  MoveL 2858 to (545.28, 463.11, 48) mm, rotated rx -180 ry 0 rz 160 deg; joints [1.397, 78.332, -23.257, -154.456, 57.789, 165.708]
  Call Extruder(423.12650)
  MoveL 2859 to (546.03, 464.05, 48) mm, rotated rx 180 ry 0 rz 160 deg; joints [1.504, 78.485, -23.584, -154.287, 57.658, 165.554]
  Set speed (17.6 mm/s)
  Call Extruder(426.93166)
  MoveL 2860 to (546.75, 464.99, 48) mm, rotated rx -180 ry 0 rz 160 deg; joints [1.61, 78.632, -23.9, -154.118, 57.533, 165.401]
  Set speed (17.6 mm/s)
  Call Extruder(430.87800)
  MoveL 2861 to (547.48, 465.98, 48) mm, rotated rx 180 ry 0 rz 160 deg; joints [1.722, 78.782, -24.221, -153.941, 57.407, 165.243]
  Set speed (17.6 mm/s)
  Call Extruder(434.56337)
  MoveL 2862 to (548.14, 466.92, 48) mm, rotated rx 180 ry 0 rz 160 deg; joints [1.828, 78.92, -24.516, -153.776, 57.293, 165.095]
  Set speed (17.6 mm/s)
  Call Extruder(438.45260)
  MoveL 2863 to (548.81, 467.93, 48) mm, rotated rx -180 ry 0 rz 160 deg; joints [1.941, 79.062, -24.821, -153.599, 57.177, 164.94]
  Set speed (17.6 mm/s)
  Call Extruder(442.25039)
  MoveL 2864 to (549.45, 468.92, 48) mm, rotated rx -180 ry 0 rz 160 deg; joints [2.053, 79.2, -25.114, -153.426, 57.067, 164.787]
  Set speed (17.6 mm/s)
  Call Extruder(446.16761)
  MoveL 2865 to (550.09, 469.96, 48) mm, rotated rx 180 ry 0 rz 160 deg; joints [2.17, 79.337, -25.408, -153.247, 56.958, 164.631]
  Set speed (17.6 mm/s)
  Call Extruder(449.89930)
  MoveL 2866 to (550.68, 470.96, 48) mm, rotated rx 180 ry 0 rz 160 deg; joints [2.282, 79.467, -25.683, -153.075, 56.857, 164.481]
  Set speed (17.6 mm/s)
  Call Extruder(454.87335)
  MoveL 2867 to (551.43, 472.32, 48) mm, rotated rx -180 ry 0 rz 160 deg; joints [2.433, 79.634, -26.039, -152.844, 56.73, 164.284]
  Call Extruder(457.60694)
  MoveL 2868 to (551.83, 473.07, 48) mm, rotated rx -180 ry 0 rz 160 deg; joints [2.517, 79.723, -26.229, -152.717, 56.664, 164.175]
  Set speed (17.6 mm/s)
  Call Extruder(461.47028)
  MoveL 2869 to (552.38, 474.15, 48) mm, rotated rx -180 ry 0 rz 160 deg; joints [2.637, 79.847, -26.493, -152.537, 56.572, 164.023]
  Call Extruder(465.26660)
  MoveL 2870 to (552.89, 475.21, 48) mm, rotated rx -180 ry 0 rz 160 deg; joints [2.756, 79.966, -26.744, -152.36, 56.487, 163.873]
  Call Extruder(469.15969)
  MoveL 2871 to (553.39, 476.32, 48) mm, rotated rx 180 ry 0 rz 160 deg; joints [2.878, 80.083, -26.994, -152.177, 56.405, 163.721]
  Set speed (17.6 mm/s)
  Call Extruder(473.03101)
  MoveL 2872 to (553.87, 477.43, 48) mm, rotated rx -180 ry 0 rz 160 deg; joints [3.002, 80.196, -27.233, -151.996, 56.328, 163.572]
  Set speed (17.6 mm/s)
  Call Extruder(476.66330)
  MoveL 2873 to (554.3, 478.47, 48) mm, rotated rx -180 ry 0 rz 160 deg; joints [3.118, 80.3, -27.453, -151.826, 56.258, 163.432]
  Set speed (17.6 mm/s)
  Call Extruder(484.36900)
  MoveL 2874 to (555.14, 480.72, 48) mm, rotated rx 180 ry 0 rz 160 deg; joints [3.367, 80.508, -27.894, -151.464, 56.126, 163.139]
  Set speed (17.6 mm/s)
  Call Extruder(488.35091)
  MoveL 2875 to (555.53, 481.9, 48) mm, rotated rx -180 ry 0 rz 160 deg; joints [3.498, 80.609, -28.106, -151.278, 56.066, 162.991]
  Set speed (17.6 mm/s)
  Call Extruder(492.11041)
  MoveL 2876 to (555.88, 483.01, 48) mm, rotated rx -180 ry 0 rz 160 deg; joints [3.621, 80.701, -28.301, -151.102, 56.012, 162.851]
  Call Extruder(496.03639)
  MoveL 2877 to (556.22, 484.19, 48) mm, rotated rx -180 ry 0 rz 160 deg; joints [3.751, 80.792, -28.492, -150.919, 55.962, 162.709]
  Set speed (17.6 mm/s)
  Call Extruder(499.92428)
  MoveL 2878 to (556.54, 485.35, 48) mm, rotated rx -180 ry 0 rz 160 deg; joints [3.881, 80.879, -28.677, -150.738, 55.916, 162.568]
  Set speed (17.6 mm/s)
  Call Extruder(507.43789)
  MoveL 2879 to (557.09, 487.63, 48) mm, rotated rx -180 ry 0 rz 160 deg; joints [4.133, 81.034, -29.003, -150.391, 55.843, 162.303]
  Set speed (17.6 mm/s)
  Call Extruder(515.16993)
  MoveL 2880 to (557.55, 490, 48) mm, rotated rx -180 ry 0 rz 160 deg; joints [4.395, 81.176, -29.302, -150.036, 55.787, 162.039]
  Set speed (17.6 mm/s)
  Call Extruder(522.84550)
  MoveL 2881 to (557.91, 492.36, 48) mm, rotated rx -180 ry 0 rz 160 deg; joints [4.658, 81.298, -29.56, -149.688, 55.751, 161.788]
  Set speed (17.6 mm/s)
  Call Extruder(530.59967)
  MoveL 2882 to (558.17, 494.77, 48) mm, rotated rx -180 ry 0 rz 160 deg; joints [4.924, 81.404, -29.781, -149.341, 55.735, 161.544]
  Set speed (17.6 mm/s)
  Call Extruder(538.17218)
  MoveL 2883 to (558.34, 497.12, 48) mm, rotated rx 180 ry 0 rz 160 deg; joints [5.187, 81.488, -29.957, -149.008, 55.74, 161.317]
  Set speed (17.6 mm/s)
  Call Extruder(545.84219)
  MoveL 2884 to (558.41, 499.51, 48) mm, rotated rx 180 ry 0 rz 160 deg; joints [5.453, 81.553, -30.096, -148.677, 55.764, 161.1]
  Set speed (17.6 mm/s)
  Call Extruder(553.37640)
  MoveL 2885 to (558.38, 501.86, 48) mm, rotated rx -180 ry 0 rz 160 deg; joints [5.716, 81.599, -30.192, -148.359, 55.806, 160.899]
  Set speed (17.6 mm/s)
  Call Extruder(561.15643)
  MoveL 2886 to (558.25, 504.28, 48) mm, rotated rx -180 ry 0 rz 160 deg; joints [5.988, 81.627, -30.25, -148.038, 55.87, 160.705]
  Set speed (17.6 mm/s)
  Call Extruder(568.72691)
  MoveL 2887 to (558.03, 506.63, 48) mm, rotated rx 180 ry 0 rz 160 deg; joints [6.253, 81.634, -30.264, -147.733, 55.951, 160.531]
  Set speed (17.6 mm/s)
  Call Extruder(576.57629)
  MoveL 2888 to (557.7, 509.06, 48) mm, rotated rx -180 ry 0 rz 160 deg; joints [6.528, 81.621, -30.238, -147.426, 56.055, 160.366]
  Set speed (17.6 mm/s)
  Call Extruder(584.14957)
  MoveL 2889 to (557.29, 511.38, 48) mm, rotated rx -180 ry 0 rz 160 deg; joints [6.793, 81.589, -30.17, -147.139, 56.174, 160.221]
  Set speed (17.6 mm/s)
  Call Extruder(591.90187)
  MoveL 2890 to (556.77, 513.74, 48) mm, rotated rx -180 ry 0 rz 160 deg; joints [7.063, 81.537, -30.061, -146.854, 56.314, 160.089]
  Call Extruder(599.47109)
  MoveL 2891 to (556.17, 516.02, 48) mm, rotated rx -180 ry 0 rz 160 deg; joints [7.326, 81.466, -29.912, -146.585, 56.469, 159.976]
  Set speed (17.6 mm/s)
  Call Extruder(602.44592)
  MoveL 2892 to (555.91, 516.91, 48) mm, rotated rx 180 ry 0 rz 160 deg; joints [7.429, 81.432, -29.841, -146.483, 56.535, 159.937]
  Set speed (17.6 mm/s)
  Call Extruder(607.08358)
  MoveL 2893 to (555.47, 518.29, 48) mm, rotated rx 180 ry 0 rz 160 deg; joints [7.588, 81.376, -29.722, -146.326, 56.642, 159.879]
  Set speed (17.6 mm/s)
  Call Extruder(614.72062)
  MoveL 2894 to (554.68, 520.53, 48) mm, rotated rx 180 ry 0 rz 160 deg; joints [7.851, 81.267, -29.494, -146.075, 56.832, 159.797]
  Set speed (17.6 mm/s)
  Call Extruder(618.66676)
  MoveL 2895 to (554.23, 521.68, 48) mm, rotated rx -180 ry 0 rz 160 deg; joints [7.986, 81.203, -29.358, -145.95, 56.937, 159.762]
  Set speed (17.6 mm/s)
  Call Extruder(622.59881)
  MoveL 2896 to (553.77, 522.81, 48) mm, rotated rx -180 ry 0 rz 160 deg; joints [8.12, 81.136, -29.218, -145.827, 57.044, 159.73]
  Set speed (17.6 mm/s)
  Call Extruder(626.34222)
  MoveL 2897 to (553.3, 523.88, 48) mm, rotated rx -180 ry 0 rz 160 deg; joints [8.246, 81.066, -29.07, -145.714, 57.152, 159.705]
  Set speed (17.6 mm/s)
  Call Extruder(630.01061)
  MoveL 2898 to (552.83, 524.92, 48) mm, rotated rx -180 ry 0 rz 160 deg; joints [8.37, 80.995, -28.921, -145.604, 57.26, 159.683]
  Set speed (17.6 mm/s)
  Call Extruder(634.07248)
  MoveL 2899 to (552.27, 526.06, 48) mm, rotated rx -180 ry 0 rz 160 deg; joints [8.506, 80.912, -28.745, -145.486, 57.384, 159.663]
  Set speed (17.6 mm/s)
  Call Extruder(638.12886)
  MoveL 2900 to (551.7, 527.18, 48) mm, rotated rx -180 ry 0 rz 160 deg; joints [8.642, 80.823, -28.559, -145.371, 57.512, 159.648]
  Call Extruder(641.69777)
  MoveL 2901 to (551.17, 528.16, 48) mm, rotated rx 180 ry 0 rz 160 deg; joints [8.76, 80.741, -28.385, -145.272, 57.628, 159.639]
  Set speed (17.6 mm/s)
  Call Extruder(645.41195)
  MoveL 2902 to (550.6, 529.17, 48) mm, rotated rx -180 ry 0 rz 160 deg; joints [8.883, 80.652, -28.198, -145.171, 57.752, 159.633]
  Set speed (17.6 mm/s)
  Call Extruder(649.34423)
  MoveL 2903 to (549.98, 530.23, 48) mm, rotated rx -180 ry 0 rz 160 deg; joints [9.012, 80.554, -27.991, -145.068, 57.886, 159.63]
  Set speed (17.6 mm/s)
  Call Extruder(653.08075)
  MoveL 2904 to (549.37, 531.22, 48) mm, rotated rx 180 ry 0 rz 160 deg; joints [9.134, 80.457, -27.785, -144.972, 58.017, 159.632]
  Set speed (17.6 mm/s)
  Call Extruder(656.63345)
  MoveL 2905 to (548.77, 532.15, 48) mm, rotated rx -180 ry 0 rz 160 deg; joints [9.249, 80.361, -27.582, -144.883, 58.145, 159.637]
  Set speed (17.6 mm/s)
  Call Extruder(660.74663)
  MoveL 2906 to (548.05, 533.21, 48) mm, rotated rx 180 ry 0 rz 160 deg; joints [9.382, 80.245, -27.338, -144.783, 58.297, 159.648]
  Set speed (17.6 mm/s)
  Call Extruder(664.63531)
  MoveL 2907 to (547.35, 534.2, 48) mm, rotated rx -180 ry 0 rz 160 deg; joints [9.506, 80.133, -27.1, -144.691, 58.442, 159.661]
  Set speed (17.6 mm/s)
  Call Extruder(668.54814)
  MoveL 2908 to (546.62, 535.19, 48) mm, rotated rx 180 ry 0 rz 160 deg; joints [9.63, 80.017, -26.853, -144.601, 58.592, 159.678]
  Call Extruder(672.23601)
  MoveL 2909 to (545.92, 536.1, 48) mm, rotated rx -180 ry 0 rz 160 deg; joints [9.746, 79.903, -26.611, -144.519, 58.736, 159.699]
  Set speed (17.6 mm/s)
  Call Extruder(676.15166)
  MoveL 2910 to (545.16, 537.05, 48) mm, rotated rx -180 ry 0 rz 160 deg; joints [9.868, 79.779, -26.348, -144.434, 58.892, 159.724]
  Call Extruder(679.91758)
  MoveL 2911 to (544.4, 537.95, 48) mm, rotated rx -180 ry 0 rz 160 deg; joints [9.984, 79.656, -26.087, -144.355, 59.044, 159.753]
  Set speed (17.6 mm/s)
  Call Extruder(683.75230)
  MoveL 2912 to (543.62, 538.85, 48) mm, rotated rx 180 ry 0 rz 160 deg; joints [10.101, 79.528, -25.815, -144.278, 59.202, 159.785]
  Call Extruder(687.54414)
  MoveL 2913 to (542.82, 539.72, 48) mm, rotated rx 180 ry 0 rz 160 deg; joints [10.216, 79.399, -25.54, -144.203, 59.36, 159.82]
  Set speed (17.6 mm/s)
  Call Extruder(690.70425)
  MoveL 2914 to (542.15, 540.44, 48) mm, rotated rx 180 ry 0 rz 160 deg; joints [10.31, 79.289, -25.305, -144.143, 59.494, 159.853]
  Set speed (17.6 mm/s)
  Call Extruder(695.32985)
  MoveL 2915 to (541.14, 541.47, 48) mm, rotated rx -180 ry 0 rz 160 deg; joints [10.447, 79.124, -24.953, -144.058, 59.692, 159.904]
  Call Extruder(699.09786)
  MoveL 2916 to (540.29, 542.28, 48) mm, rotated rx 180 ry 0 rz 160 deg; joints [10.557, 78.987, -24.66, -143.992, 59.856, 159.95]
  Set speed (17.6 mm/s)
  Call Extruder(702.88058)
  MoveL 2917 to (539.43, 543.09, 48) mm, rotated rx -180 ry 0 rz 160 deg; joints [10.666, 78.846, -24.359, -143.928, 60.023, 160]
  Set speed (17.6 mm/s)
  Call Extruder(706.79322)
  MoveL 2918 to (538.52, 543.9, 48) mm, rotated rx 180 ry 0 rz 160 deg; joints [10.778, 78.698, -24.042, -143.864, 60.198, 160.054]
  Set speed (17.6 mm/s)
  Call Extruder(710.57041)
  MoveL 2919 to (537.63, 544.67, 48) mm, rotated rx -180 ry 0 rz 160 deg; joints [10.885, 78.553, -23.731, -143.804, 60.368, 160.11]
  Set speed (17.6 mm/s)
  Call Extruder(717.12256)
  MoveL 2920 to (536.05, 545.96, 48) mm, rotated rx 180 ry 0 rz 160 deg; joints [11.066, 78.296, -23.178, -143.707, 60.668, 160.214]
  Call Extruder(722.16766)
  MoveL 2921 to (534.8, 546.92, 48) mm, rotated rx 180 ry 0 rz 160 deg; joints [11.203, 78.093, -22.743, -143.637, 60.902, 160.3]
  Set speed (17.6 mm/s)
  Call Extruder(725.90272)
  MoveL 2922 to (533.85, 547.6, 48) mm, rotated rx -180 ry 0 rz 160 deg; joints [11.302, 77.94, -22.413, -143.588, 61.077, 160.368]
  Call Extruder(729.71251)
  MoveL 2923 to (532.88, 548.28, 48) mm, rotated rx 180 ry 0 rz 160 deg; joints [11.402, 77.783, -22.074, -143.54, 61.257, 160.439]
  Set speed (17.6 mm/s)
  Call Extruder(733.60669)
  MoveL 2924 to (531.87, 548.95, 48) mm, rotated rx -180 ry 0 rz 160 deg; joints [11.502, 77.62, -21.723, -143.494, 61.442, 160.516]
  Set speed (17.6 mm/s)
  Call Extruder(737.39555)
  MoveL 2925 to (530.87, 549.59, 48) mm, rotated rx 180 ry 0 rz 160 deg; joints [11.598, 77.46, -21.376, -143.451, 61.624, 160.593]
  Set speed (17.6 mm/s)
  Call Extruder(741.30942)
  MoveL 2926 to (529.83, 550.22, 48) mm, rotated rx -180 ry 0 rz 160 deg; joints [11.695, 77.293, -21.015, -143.409, 61.812, 160.675]
  Set speed (17.6 mm/s)
  Call Extruder(745.06218)
  MoveL 2927 to (528.82, 550.81, 48) mm, rotated rx -180 ry 0 rz 160 deg; joints [11.787, 77.131, -20.663, -143.372, 61.994, 160.757]
  Call Extruder(748.32344)
  MoveL 2928 to (527.93, 551.3, 48) mm, rotated rx 180 ry 0 rz 160 deg; joints [11.865, 76.989, -20.356, -143.34, 62.153, 160.829]
  Call Extruder(752.73182)
  MoveL 2929 to (526.72, 551.94, 48) mm, rotated rx 180 ry 0 rz 160 deg; joints [11.968, 76.795, -19.935, -143.302, 62.369, 160.931]
  Call Extruder(756.56366)
  MoveL 2930 to (525.65, 552.48, 48) mm, rotated rx -180 ry 0 rz 160 deg; joints [12.056, 76.626, -19.566, -143.27, 62.558, 161.023]
  Set speed (17.6 mm/s)
  Call Extruder(760.56830)
  MoveL 2931 to (524.52, 553.01, 48) mm, rotated rx -180 ry 0 rz 160 deg; joints [12.146, 76.447, -19.176, -143.24, 62.756, 161.121]
  Set speed (17.6 mm/s)
  Call Extruder(764.31154)
  MoveL 2932 to (523.46, 553.49, 48) mm, rotated rx 180 ry 0 rz 160 deg; joints [12.227, 76.279, -18.808, -143.214, 62.942, 161.215]
  Set speed (17.6 mm/s)
  Call Extruder(768.13737)
  MoveL 2933 to (522.36, 553.96, 48) mm, rotated rx -180 ry 0 rz 160 deg; joints [12.309, 76.107, -18.432, -143.189, 63.132, 161.313]
  Set speed (17.6 mm/s)
  Call Extruder(775.62142)
  MoveL 2934 to (520.19, 554.81, 48) mm, rotated rx 180 ry 0 rz 160 deg; joints [12.463, 75.765, -17.685, -143.148, 63.506, 161.512]
  Set speed (17.6 mm/s)
  Call Extruder(779.70711)
  MoveL 2935 to (518.99, 555.23, 48) mm, rotated rx -180 ry 0 rz 160 deg; joints [12.544, 75.578, -17.273, -143.13, 63.711, 161.625]
  Set speed (17.6 mm/s)
  Call Extruder(783.37834)
  MoveL 2936 to (517.91, 555.6, 48) mm, rotated rx -180 ry 0 rz 160 deg; joints [12.614, 75.41, -16.903, -143.115, 63.895, 161.727]
  Set speed (17.6 mm/s)
  Call Extruder(787.32169)
  MoveL 2937 to (516.73, 555.95, 48) mm, rotated rx 180 ry 0 rz 160 deg; joints [12.687, 75.227, -16.5, -143.102, 64.093, 161.84]
  Set speed (17.6 mm/s)
  Call Extruder(791.11815)
  MoveL 2938 to (515.6, 556.29, 48) mm, rotated rx -180 ry 0 rz 160 deg; joints [12.756, 75.052, -16.113, -143.091, 64.284, 161.949]
  Set speed (17.6 mm/s)
  Call Extruder(795.03560)
  MoveL 2939 to (514.42, 556.6, 48) mm, rotated rx 180 ry 0 rz 160 deg; joints [12.824, 74.869, -15.71, -143.083, 64.481, 162.066]
  Call Extruder(798.82897)
  MoveL 2940 to (513.27, 556.88, 48) mm, rotated rx -180 ry 0 rz 160 deg; joints [12.888, 74.693, -15.32, -143.076, 64.672, 162.179]
  Set speed (17.6 mm/s)
  Call Extruder(806.50817)
  MoveL 2941 to (510.93, 557.38, 48) mm, rotated rx -180 ry 0 rz 160 deg; joints [13.01, 74.334, -14.523, -143.071, 65.059, 162.415]
  Set speed (17.6 mm/s)
  Call Extruder(814.22140)
  MoveL 2942 to (508.56, 557.78, 48) mm, rotated rx 180 ry 0 rz 160 deg; joints [13.123, 73.973, -13.719, -143.076, 65.448, 162.658]
  Set speed (17.6 mm/s)
  Call Extruder(821.72414)
  MoveL 2943 to (506.24, 558.07, 48) mm, rotated rx 180 ry 0 rz 160 deg; joints [13.222, 73.622, -12.933, -143.09, 65.824, 162.902]
  Set speed (17.6 mm/s)
  Call Extruder(829.51820)
  MoveL 2944 to (503.82, 558.28, 48) mm, rotated rx 180 ry 0 rz 160 deg; joints [13.316, 73.258, -12.116, -143.113, 66.214, 163.16]
  Set speed (17.6 mm/s)
  Call Extruder(837.23307)
  MoveL 2945 to (501.42, 558.39, 48) mm, rotated rx -180 ry 0 rz 160 deg; joints [13.397, 72.898, -11.306, -143.146, 66.598, 163.421]
  Set speed (17.6 mm/s)
  Call Extruder(844.81348)
  MoveL 2946 to (499.05, 558.4, 48) mm, rotated rx -180 ry 0 rz 160 deg; joints [13.467, 72.546, -10.51, -143.188, 66.972, 163.682]
  Set speed (10.0 mm/s)
  MoveL 2947 to (499.05, 558.4, 52) mm, rotated rx 180 ry 0 rz 160 deg; joints [13.467, 71.85, -10.06, -143.125, 66.776, 163.521]
  Set speed (120.0 mm/s)
  MoveL 2948 to (499.05, 559.26, 52) mm, rotated rx 180 ry 0 rz 160 deg; joints [13.571, 71.88, -10.127, -143.006, 66.775, 163.454]
  Set speed (17.6 mm/s)
  Call Extruder(852.64361)
  MoveL 2949 to (496.6, 559.17, 52) mm, rotated rx 180 ry 0 rz 160 deg; joints [13.631, 71.517, -9.309, -143.06, 67.157, 163.728]
  Set speed (17.6 mm/s)
  Call Extruder(860.45123)
  MoveL 2950 to (494.17, 558.98, 52) mm, rotated rx -180 ry 0 rz 160 deg; joints [13.68, 71.159, -8.496, -143.123, 67.534, 164.003]
  Set speed (17.6 mm/s)
  Call Extruder(868.29937)
  MoveL 2951 to (491.74, 558.69, 52) mm, rotated rx -180 ry 0 rz 160 deg; joints [13.717, 70.802, -7.684, -143.197, 67.908, 164.284]
  Call Extruder(875.80436)
  MoveL 2952 to (489.43, 558.32, 52) mm, rotated rx 180 ry 0 rz 160 deg; joints [13.741, 70.465, -6.912, -143.276, 68.262, 164.555]
  Set speed (17.6 mm/s)
  Call Extruder(883.78153)
  MoveL 2953 to (486.99, 557.82, 52) mm, rotated rx -180 ry 0 rz 160 deg; joints [13.753, 70.11, -6.099, -143.372, 68.634, 164.845]
  Set speed (17.6 mm/s)
  Call Extruder(887.61260)
  MoveL 2954 to (485.83, 557.54, 52) mm, rotated rx -180 ry 0 rz 160 deg; joints [13.754, 69.942, -5.711, -143.422, 68.81, 164.985]
  Set speed (17.6 mm/s)
  Call Extruder(891.58436)
  MoveL 2955 to (484.63, 557.24, 52) mm, rotated rx 180 ry 0 rz 160 deg; joints [13.753, 69.769, -5.311, -143.475, 68.992, 165.13]
  Set speed (17.6 mm/s)
  Call Extruder(899.15379)
  MoveL 2956 to (482.36, 556.58, 52) mm, rotated rx -180 ry 0 rz 160 deg; joints [13.74, 69.442, -4.555, -143.586, 69.334, 165.408]
  Set speed (17.6 mm/s)
  Call Extruder(903.12349)
  MoveL 2957 to (481.19, 556.2, 52) mm, rotated rx -180 ry 0 rz 160 deg; joints [13.727, 69.273, -4.162, -143.648, 69.511, 165.554]
  Set speed (17.6 mm/s)
  Call Extruder(906.96713)
  MoveL 2958 to (480.05, 555.81, 52) mm, rotated rx 180 ry 0 rz 160 deg; joints [13.714, 69.111, -3.784, -143.71, 69.681, 165.695]
  Set speed (17.6 mm/s)
  Call Extruder(910.94545)
  MoveL 2959 to (478.89, 555.38, 52) mm, rotated rx -180 ry 0 rz 160 deg; joints [13.695, 68.944, -3.396, -143.778, 69.855, 165.842]
  Set speed (17.6 mm/s)
  Call Extruder(914.78044)
  MoveL 2960 to (477.78, 554.95, 52) mm, rotated rx -180 ry 0 rz 160 deg; joints [13.674, 68.785, -3.024, -143.845, 70.022, 165.983]
  Set speed (17.6 mm/s)
  Call Extruder(920.70005)
  MoveL 2961 to (476.08, 554.23, 52) mm, rotated rx 180 ry 0 rz 160 deg; joints [13.636, 68.543, -2.457, -143.954, 70.276, 166.2]
  Call Extruder(922.64903)
  MoveL 2962 to (475.52, 553.98, 52) mm, rotated rx 180 ry 0 rz 160 deg; joints [13.621, 68.464, -2.271, -143.991, 70.358, 166.272]
  Set speed (17.6 mm/s)
  Call Extruder(926.38246)
  MoveL 2963 to (474.47, 553.49, 52) mm, rotated rx 180 ry 0 rz 160 deg; joints [13.591, 68.314, -1.918, -144.065, 70.516, 166.409]
  Call Extruder(930.30379)
  MoveL 2964 to (473.37, 552.95, 52) mm, rotated rx 180 ry 0 rz 160 deg; joints [13.556, 68.158, -1.55, -144.145, 70.68, 166.553]
  Call Extruder(934.18803)
  MoveL 2965 to (472.29, 552.4, 52) mm, rotated rx 180 ry 0 rz 160 deg; joints [13.518, 68.005, -1.188, -144.226, 70.84, 166.695]
  Set speed (17.6 mm/s)
  Call Extruder(938.04188)
  MoveL 2966 to (471.24, 551.82, 52) mm, rotated rx -180 ry 0 rz 160 deg; joints [13.477, 67.855, -0.833, -144.31, 70.997, 166.835]
  Set speed (17.6 mm/s)
  Call Extruder(941.96003)
  MoveL 2967 to (470.17, 551.22, 52) mm, rotated rx 180 ry 0 rz 160 deg; joints [13.432, 67.704, -0.476, -144.398, 71.155, 166.978]
  Call Extruder(945.88432)
  MoveL 2968 to (469.12, 550.59, 52) mm, rotated rx 180 ry 0 rz 160 deg; joints [13.383, 67.556, -0.122, -144.489, 71.311, 167.12]
  Set speed (17.6 mm/s)
  Call Extruder(949.75357)
  MoveL 2969 to (468.1, 549.95, 52) mm, rotated rx 180 ry 0 rz 160 deg; joints [13.332, 67.411, 0.224, -144.581, 71.463, 167.26]
  Call Extruder(953.68094)
  MoveL 2970 to (467.07, 549.28, 52) mm, rotated rx -180 ry 0 rz 160 deg; joints [13.276, 67.266, 0.57, -144.677, 71.615, 167.401]
  Set speed (17.6 mm/s)
  Call Extruder(957.51292)
  MoveL 2971 to (466.08, 548.6, 52) mm, rotated rx 180 ry 0 rz 160 deg; joints [13.218, 67.126, 0.904, -144.774, 71.761, 167.538]
  Call Extruder(961.37055)
  MoveL 2972 to (465.1, 547.9, 52) mm, rotated rx -180 ry 0 rz 160 deg; joints [13.157, 66.988, 1.236, -144.874, 71.906, 167.675]
  Set speed (17.6 mm/s)
  Call Extruder(965.21214)
  MoveL 2973 to (464.14, 547.19, 52) mm, rotated rx 180 ry 0 rz 160 deg; joints [13.092, 66.852, 1.563, -144.976, 72.049, 167.811]
  Set speed (17.6 mm/s)
  Call Extruder(969.14916)
  MoveL 2974 to (463.17, 546.44, 52) mm, rotated rx -180 ry 0 rz 160 deg; joints [13.023, 66.715, 1.893, -145.083, 72.193, 167.95]
  Set speed (17.6 mm/s)
  Call Extruder(973.20799)
  MoveL 2975 to (462.18, 545.64, 52) mm, rotated rx -180 ry 0 rz 160 deg; joints [12.947, 66.577, 2.229, -145.196, 72.339, 168.091]
  Set speed (17.6 mm/s)
  Call Extruder(976.91657)
  MoveL 2976 to (461.3, 544.89, 52) mm, rotated rx -180 ry 0 rz 160 deg; joints [12.875, 66.452, 2.531, -145.302, 72.469, 168.22]
  Set speed (17.6 mm/s)
  Call Extruder(980.80542)
  MoveL 2977 to (460.39, 544.09, 52) mm, rotated rx -180 ry 0 rz 160 deg; joints [12.796, 66.323, 2.843, -145.416, 72.604, 168.353]
  Set speed (17.6 mm/s)
  Call Extruder(986.38850)
  MoveL 2978 to (459.11, 542.91, 52) mm, rotated rx 180 ry 0 rz 160 deg; joints [12.678, 66.142, 3.284, -145.584, 72.795, 168.544]
  Set speed (17.6 mm/s)
  Call Extruder(992.43638)
  MoveL 2979 to (457.76, 541.58, 52) mm, rotated rx 180 ry 0 rz 160 deg; joints [12.54, 65.952, 3.748, -145.772, 72.994, 168.747]
  Set speed (17.6 mm/s)
  Call Extruder(996.28555)
  MoveL 2980 to (456.93, 540.72, 52) mm, rotated rx 180 ry 0 rz 160 deg; joints [12.449, 65.834, 4.037, -145.895, 73.118, 168.875]
  Set speed (17.6 mm/s)
  Call Extruder(1000.06433)
  MoveL 2981 to (456.13, 539.85, 52) mm, rotated rx 180 ry 0 rz 160 deg; joints [12.356, 65.721, 4.316, -146.018, 73.237, 168.999]
  Call Extruder(1004.06459)
  MoveL 2982 to (455.3, 538.92, 52) mm, rotated rx 180 ry 0 rz 160 deg; joints [12.254, 65.603, 4.605, -146.151, 73.36, 169.129]
  Set speed (17.6 mm/s)
  Call Extruder(1007.98301)
  MoveL 2983 to (454.51, 537.99, 52) mm, rotated rx -180 ry 0 rz 160 deg; joints [12.152, 65.49, 4.883, -146.284, 73.478, 169.255]
  Call Extruder(1011.82469)
  MoveL 2984 to (453.75, 537.06, 52) mm, rotated rx 180 ry 0 rz 160 deg; joints [12.047, 65.382, 5.15, -146.417, 73.591, 169.377]
  Call Extruder(1015.92450)
  MoveL 2985 to (452.96, 536.05, 52) mm, rotated rx -180 ry 0 rz 160 deg; joints [11.933, 65.269, 5.43, -146.56, 73.71, 169.506]
  Call Extruder(1019.64122)
  MoveL 2986 to (452.26, 535.12, 52) mm, rotated rx -180 ry 0 rz 160 deg; joints [11.827, 65.169, 5.677, -146.693, 73.813, 169.621]
  Set speed (17.6 mm/s)
  Call Extruder(1023.51639)
  MoveL 2987 to (451.55, 534.14, 52) mm, rotated rx -180 ry 0 rz 160 deg; joints [11.713, 65.068, 5.93, -146.834, 73.919, 169.739]
  Set speed (17.6 mm/s)
  Call Extruder(1026.78205)
  MoveL 2988 to (450.98, 533.3, 52) mm, rotated rx -180 ry 0 rz 160 deg; joints [11.614, 64.985, 6.137, -146.955, 74.006, 169.838]
  Call Extruder(1031.07858)
  MoveL 2989 to (450.23, 532.19, 52) mm, rotated rx -180 ry 0 rz 160 deg; joints [11.481, 64.878, 6.404, -147.116, 74.117, 169.966]
  Set speed (17.6 mm/s)
  Call Extruder(1035.12806)
  MoveL 2990 to (449.56, 531.12, 52) mm, rotated rx 180 ry 0 rz 160 deg; joints [11.353, 64.779, 6.649, -147.27, 74.218, 170.084]
  Set speed (17.6 mm/s)
  Call Extruder(1039.06221)
  MoveL 2991 to (448.92, 530.07, 52) mm, rotated rx 180 ry 0 rz 160 deg; joints [11.225, 64.687, 6.881, -147.422, 74.313, 170.198]
  Set speed (17.6 mm/s)
  Call Extruder(1042.92344)
  MoveL 2992 to (448.32, 529.03, 52) mm, rotated rx 180 ry 0 rz 160 deg; joints [11.097, 64.599, 7.102, -147.573, 74.404, 170.307]
  Set speed (17.6 mm/s)
  Call Extruder(1046.81692)
  MoveL 2993 to (447.74, 527.96, 52) mm, rotated rx -180 ry 0 rz 160 deg; joints [10.964, 64.513, 7.318, -147.728, 74.491, 170.416]
  Call Extruder(1050.65850)
  MoveL 2994 to (447.19, 526.9, 52) mm, rotated rx 180 ry 0 rz 160 deg; joints [10.831, 64.431, 7.526, -147.882, 74.575, 170.521]
  Set speed (17.6 mm/s)
  Call Extruder(1054.63199)
  MoveL 2995 to (446.64, 525.79, 52) mm, rotated rx 180 ry 0 rz 160 deg; joints [10.691, 64.349, 7.733, -148.044, 74.658, 170.628]
  Set speed (17.6 mm/s)
  Call Extruder(1058.58359)
  MoveL 2996 to (446.12, 524.67, 52) mm, rotated rx 180 ry 0 rz 160 deg; joints [10.548, 64.27, 7.931, -148.207, 74.737, 170.733]
  Set speed (17.6 mm/s)
  Call Extruder(1062.27178)
  MoveL 2997 to (445.64, 523.62, 52) mm, rotated rx -180 ry 0 rz 160 deg; joints [10.414, 64.198, 8.113, -148.361, 74.809, 170.829]
  Set speed (17.6 mm/s)
  Call Extruder(1070.02259)
  MoveL 2998 to (444.72, 521.38, 52) mm, rotated rx -180 ry 0 rz 160 deg; joints [10.122, 64.057, 8.471, -148.689, 74.948, 171.024]
  Set speed (17.6 mm/s)
  Call Extruder(1074.13716)
  MoveL 2999 to (444.28, 520.18, 52) mm, rotated rx 180 ry 0 rz 160 deg; joints [9.964, 63.987, 8.649, -148.867, 75.016, 171.124]
  Set speed (17.6 mm/s)
  Call Extruder(1077.86962)
  MoveL 3000 to (443.89, 519.09, 52) mm, rotated rx -180 ry 0 rz 160 deg; joints [9.818, 63.926, 8.806, -149.028, 75.075, 171.213]
  Call Extruder(1081.89672)
  MoveL 3001 to (443.5, 517.89, 52) mm, rotated rx -180 ry 0 rz 160 deg; joints [9.659, 63.863, 8.965, -149.205, 75.134, 171.307]
  Set speed (17.6 mm/s)
  Call Extruder(1085.57261)
  MoveL 3002 to (443.16, 516.8, 52) mm, rotated rx 180 ry 0 rz 160 deg; joints [9.512, 63.808, 9.107, -149.367, 75.186, 171.391]
  Set speed (17.6 mm/s)
  Call Extruder(1089.66403)
  MoveL 3003 to (442.82, 515.57, 52) mm, rotated rx 180 ry 0 rz 160 deg; joints [9.345, 63.75, 9.254, -149.55, 75.239, 171.481]
  Call Extruder(1093.47837)
  MoveL 3004 to (442.51, 514.42, 52) mm, rotated rx -180 ry 0 rz 160 deg; joints [9.189, 63.698, 9.387, -149.72, 75.286, 171.564]
  Set speed (17.6 mm/s)
  Call Extruder(1096.84078)
  MoveL 3005 to (442.27, 513.4, 52) mm, rotated rx 180 ry 0 rz 160 deg; joints [9.049, 63.656, 9.496, -149.872, 75.323, 171.635]
  Set speed (17.6 mm/s)
  Call Extruder(1101.91827)
  MoveL 3006 to (441.93, 511.86, 52) mm, rotated rx 180 ry 0 rz 160 deg; joints [8.836, 63.595, 9.653, -150.102, 75.375, 171.74]
  Set speed (17.6 mm/s)
  Call Extruder(1109.14695)
  MoveL 3007 to (441.52, 509.64, 52) mm, rotated rx 180 ry 0 rz 160 deg; joints [8.527, 63.517, 9.853, -150.434, 75.437, 171.882]
  Set speed (17.6 mm/s)
  Call Extruder(1116.90127)
  MoveL 3008 to (441.17, 507.24, 52) mm, rotated rx 180 ry 0 rz 160 deg; joints [8.191, 63.444, 10.04, -150.793, 75.49, 172.026]
  Set speed (17.6 mm/s)
  Call Extruder(1124.67746)
  MoveL 3009 to (440.93, 504.83, 52) mm, rotated rx -180 ry 0 rz 160 deg; joints [7.848, 63.384, 10.197, -151.155, 75.527, 172.162]
  Set speed (17.6 mm/s)
  Call Extruder(1132.27890)
  MoveL 3010 to (440.78, 502.46, 52) mm, rotated rx 180 ry 0 rz 160 deg; joints [7.509, 63.336, 10.321, -151.511, 75.548, 172.286]
  Set speed (17.6 mm/s)
  Call Extruder(1140.11948)
  MoveL 3011 to (440.73, 500.01, 52) mm, rotated rx 180 ry 0 rz 160 deg; joints [7.157, 63.298, 10.419, -151.879, 75.554, 172.406]
  Set speed (17.6 mm/s)
  Call Extruder(1147.18943)
  MoveL 3012 to (440.77, 497.81, 52) mm, rotated rx -180 ry 0 rz 160 deg; joints [6.837, 63.274, 10.48, -152.212, 75.545, 172.506]
  Set speed (17.6 mm/s)
  Call Extruder(1154.10655)
  MoveL 3013 to (440.89, 495.65, 52) mm, rotated rx 180 ry 0 rz 160 deg; joints [6.522, 63.26, 10.516, -152.536, 75.523, 172.597]
  Set speed (17.6 mm/s)
  Call Extruder(1160.97918)
  MoveL 3014 to (441.09, 493.52, 52) mm, rotated rx 180 ry 0 rz 160 deg; joints [6.209, 63.256, 10.527, -152.858, 75.489, 172.68]
  Set speed (17.6 mm/s)
  Call Extruder(1168.08842)
  MoveL 3015 to (441.37, 491.32, 52) mm, rotated rx 180 ry 0 rz 160 deg; joints [5.886, 63.261, 10.513, -153.188, 75.441, 172.759]
  Call Extruder(1175.15451)
  MoveL 3016 to (441.74, 489.14, 52) mm, rotated rx -180 ry 0 rz 160 deg; joints [5.565, 63.276, 10.475, -153.514, 75.379, 172.831]
  Set speed (17.6 mm/s)
  Call Extruder(1182.30610)
  MoveL 3017 to (442.19, 486.95, 52) mm, rotated rx 180 ry 0 rz 160 deg; joints [5.241, 63.301, 10.409, -153.841, 75.303, 172.897]
  Set speed (17.6 mm/s)
  Call Extruder(1189.05565)
  MoveL 3018 to (442.68, 484.91, 52) mm, rotated rx 180 ry 0 rz 160 deg; joints [4.938, 63.334, 10.325, -154.147, 75.219, 172.953]
  Set speed (17.6 mm/s)
  Call Extruder(1195.93726)
  MoveL 3019 to (443.27, 482.84, 52) mm, rotated rx -180 ry 0 rz 160 deg; joints [4.631, 63.377, 10.213, -154.454, 75.12, 173.003]
  Set speed (17.6 mm/s)
  Call Extruder(1202.97463)
  MoveL 3020 to (443.95, 480.75, 52) mm, rotated rx 180 ry 0 rz 160 deg; joints [4.32, 63.431, 10.075, -154.763, 75.006, 173.047]
  Set speed (17.6 mm/s)
  Call Extruder(1209.95833)
  MoveL 3021 to (444.69, 478.7, 52) mm, rotated rx 180 ry 0 rz 160 deg; joints [4.016, 63.493, 9.914, -155.065, 74.88, 173.085]
  Set speed (17.6 mm/s)
  Call Extruder(1217.10869)
  MoveL 3022 to (445.53, 476.63, 52) mm, rotated rx -180 ry 0 rz 160 deg; joints [3.709, 63.567, 9.725, -155.368, 74.738, 173.118]
  Set speed (17.6 mm/s)
  Call Extruder(1224.00946)
  MoveL 3023 to (446.42, 474.67, 52) mm, rotated rx -180 ry 0 rz 160 deg; joints [3.417, 63.647, 9.518, -155.654, 74.588, 173.143]
  Set speed (17.6 mm/s)
  Call Extruder(1231.08379)
  MoveL 3024 to (447.4, 472.69, 52) mm, rotated rx -180 ry 0 rz 160 deg; joints [3.124, 63.739, 9.283, -155.94, 74.422, 173.163]
  Set speed (17.6 mm/s)
  Call Extruder(1237.90955)
  MoveL 3025 to (448.41, 470.82, 52) mm, rotated rx -180 ry 0 rz 160 deg; joints [2.847, 63.837, 9.033, -156.208, 74.25, 173.176]
  Set speed (17.6 mm/s)
  Call Extruder(1245.01549)
  MoveL 3026 to (449.54, 468.91, 52) mm, rotated rx -180 ry 0 rz 160 deg; joints [2.565, 63.948, 8.749, -156.479, 74.058, 173.183]
  Set speed (17.6 mm/s)
  Call Extruder(1251.96311)
  MoveL 3027 to (450.71, 467.08, 52) mm, rotated rx 180 ry 0 rz 160 deg; joints [2.297, 64.066, 8.449, -156.736, 73.86, 173.185]
  Set speed (17.6 mm/s)
  Call Extruder(1258.95622)
  MoveL 3028 to (451.96, 465.29, 52) mm, rotated rx -180 ry 0 rz 160 deg; joints [2.034, 64.194, 8.125, -156.985, 73.648, 173.18]
  Call Extruder(1266.03828)
  MoveL 3029 to (453.29, 463.52, 52) mm, rotated rx -180 ry 0 rz 160 deg; joints [1.776, 64.332, 7.774, -157.228, 73.422, 173.17]
  Set speed (17.6 mm/s)
  Call Extruder(1272.88397)
  MoveL 3030 to (454.63, 461.87, 52) mm, rotated rx -180 ry 0 rz 160 deg; joints [1.535, 64.475, 7.414, -157.453, 73.192, 173.154]
  Call Extruder(1279.93386)
  MoveL 3031 to (456.08, 460.21, 52) mm, rotated rx -180 ry 0 rz 160 deg; joints [1.295, 64.631, 7.023, -157.674, 72.946, 173.133]
  Set speed (17.6 mm/s)
  Call Extruder(1287.00387)
  MoveL 3032 to (457.59, 458.6, 52) mm, rotated rx -180 ry 0 rz 160 deg; joints [1.064, 64.795, 6.61, -157.886, 72.688, 173.105]
  Call Extruder(1293.89606)
  MoveL 3033 to (459.12, 457.09, 52) mm, rotated rx 180 ry 0 rz 160 deg; joints [0.848, 64.965, 6.186, -158.08, 72.427, 173.073]
  Set speed (17.6 mm/s)
  Call Extruder(1300.89711)
  MoveL 3034 to (460.73, 455.61, 52) mm, rotated rx -180 ry 0 rz 160 deg; joints [0.638, 65.145, 5.738, -158.267, 72.153, 173.035]
  Set speed (17.6 mm/s)
  Call Extruder(1307.97213)
  MoveL 3035 to (462.41, 454.18, 52) mm, rotated rx 180 ry 0 rz 160 deg; joints [0.436, 65.336, 5.265, -158.444, 71.866, 172.99]
  Call Extruder(1314.88669)
  MoveL 3036 to (464.1, 452.84, 52) mm, rotated rx 180 ry 0 rz 160 deg; joints [0.249, 65.53, 4.784, -158.605, 71.576, 172.941]
  Set speed (17.6 mm/s)
  Call Extruder(1321.95796)
  MoveL 3037 to (465.88, 451.53, 52) mm, rotated rx 180 ry 0 rz 160 deg; joints [0.068, 65.737, 4.275, -158.758, 71.272, 172.886]
  Set speed (17.6 mm/s)
  Call Extruder(1328.86472)
  MoveL 3038 to (467.67, 450.33, 52) mm, rotated rx 180 ry 0 rz 160 deg; joints [-0.098, 65.947, 3.76, -158.894, 70.967, 172.826]
  Call Extruder(1335.94504)
  MoveL 3039 to (469.54, 449.16, 52) mm, rotated rx -180 ry 0 rz 160 deg; joints [-0.258, 66.17, 3.215, -159.022, 70.647, 172.759]
  Call Extruder(1342.78526)
  MoveL 3040 to (471.39, 448.09, 52) mm, rotated rx -180 ry 0 rz 160 deg; joints [-0.402, 66.393, 2.673, -159.132, 70.331, 172.688]
  Set speed (17.6 mm/s)
  Call Extruder(1349.82828)
  MoveL 3041 to (473.34, 447.07, 52) mm, rotated rx -180 ry 0 rz 160 deg; joints [-0.539, 66.63, 2.1, -159.234, 69.999, 172.61]
  Call Extruder(1356.92068)
  MoveL 3042 to (475.33, 446.11, 52) mm, rotated rx 180 ry 0 rz 160 deg; joints [-0.665, 66.875, 1.507, -159.323, 69.658, 172.525]
  Set speed (17.6 mm/s)
  Call Extruder(1363.90955)
  MoveL 3043 to (477.33, 445.24, 52) mm, rotated rx 180 ry 0 rz 160 deg; joints [-0.78, 67.124, 0.909, -159.397, 69.316, 172.436]
  Set speed (17.6 mm/s)
  Call Extruder(1370.75331)
  MoveL 3044 to (479.32, 444.46, 52) mm, rotated rx -180 ry 0 rz 160 deg; joints [-0.88, 67.375, 0.31, -159.457, 68.976, 172.343]
  Set speed (17.6 mm/s)
  Call Extruder(1377.90422)
  MoveL 3045 to (481.42, 443.72, 52) mm, rotated rx 180 ry 0 rz 160 deg; joints [-0.974, 67.643, -0.329, -159.507, 68.616, 172.24]
  Set speed (17.6 mm/s)
  Call Extruder(1384.86346)
  MoveL 3046 to (483.5, 443.07, 52) mm, rotated rx -180 ry 0 rz 160 deg; joints [-1.055, 67.91, -0.963, -159.542, 68.261, 172.133]
  Set speed (17.6 mm/s)
  Call Extruder(1391.79293)
  MoveL 3047 to (485.58, 442.51, 52) mm, rotated rx -180 ry 0 rz 160 deg; joints [-1.124, 68.182, -1.606, -159.564, 67.904, 172.021]
  Set speed (17.6 mm/s)
  Call Extruder(1398.86813)
  MoveL 3048 to (487.74, 442.02, 52) mm, rotated rx 180 ry 0 rz 160 deg; joints [-1.183, 68.465, -2.274, -159.572, 67.535, 171.9]
  Set speed (17.6 mm/s)
  Call Extruder(1405.71108)
  MoveL 3049 to (489.83, 441.61, 52) mm, rotated rx 180 ry 0 rz 160 deg; joints [-1.23, 68.745, -2.93, -159.568, 67.176, 171.777]
  Set speed (17.6 mm/s)
  Call Extruder(1412.83391)
  MoveL 3050 to (492.03, 441.27, 52) mm, rotated rx -180 ry 0 rz 160 deg; joints [-1.269, 69.041, -3.622, -159.55, 66.8, 171.643]
  Call Extruder(1419.79944)
  MoveL 3051 to (494.19, 441.02, 52) mm, rotated rx -180 ry 0 rz 160 deg; joints [-1.295, 69.335, -4.308, -159.52, 66.429, 171.506]
  Set speed (17.6 mm/s)
  Call Extruder(1426.75563)
  MoveL 3052 to (496.35, 440.85, 52) mm, rotated rx 180 ry 0 rz 160 deg; joints [-1.311, 69.634, -5, -159.476, 66.058, 171.362]
  Call Extruder(1433.83398)
  MoveL 3053 to (498.56, 440.75, 52) mm, rotated rx 180 ry 0 rz 160 deg; joints [-1.317, 69.943, -5.713, -159.419, 65.679, 171.209]
  Set speed (17.6 mm/s)
  Call Extruder(1440.75355)
  MoveL 3054 to (500.72, 440.74, 52) mm, rotated rx 180 ry 0 rz 160 deg; joints [-1.312, 70.248, -6.415, -159.35, 65.308, 171.053]
  Call Extruder(1447.80768)
  MoveL 3055 to (502.92, 440.8, 52) mm, rotated rx -180 ry 0 rz 160 deg; joints [-1.297, 70.563, -7.137, -159.267, 64.93, 170.888]
  Set speed (17.6 mm/s)
  Call Extruder(1454.73515)
  MoveL 3056 to (505.08, 440.95, 52) mm, rotated rx 180 ry 0 rz 160 deg; joints [-1.273, 70.876, -7.851, -159.173, 64.558, 170.719]
  Call Extruder(1461.79106)
  MoveL 3057 to (507.27, 441.18, 52) mm, rotated rx 180 ry 0 rz 160 deg; joints [-1.238, 71.197, -8.583, -159.065, 64.181, 170.54]
  Set speed (17.6 mm/s)
  Call Extruder(1468.63957)
  MoveL 3058 to (509.39, 441.48, 52) mm, rotated rx 180 ry 0 rz 160 deg; joints [-1.194, 71.512, -9.295, -158.947, 63.816, 170.361]
  Call Extruder(1475.68058)
  MoveL 3059 to (511.55, 441.87, 52) mm, rotated rx 180 ry 0 rz 160 deg; joints [-1.14, 71.837, -10.03, -158.815, 63.443, 170.169]
  Set speed (17.6 mm/s)
  Call Extruder(1482.10061)
  MoveL 3060 to (513.51, 442.29, 52) mm, rotated rx 180 ry 0 rz 160 deg; joints [-1.084, 72.135, -10.702, -158.684, 63.105, 169.99]
  Set speed (17.6 mm/s)
  Call Extruder(1489.60636)
  MoveL 3061 to (515.78, 442.87, 52) mm, rotated rx -180 ry 0 rz 160 deg; joints [-1.007, 72.485, -11.488, -158.518, 62.713, 169.773]
  Set speed (17.6 mm/s)
  Call Extruder(1496.53533)
  MoveL 3062 to (517.85, 443.48, 52) mm, rotated rx 180 ry 0 rz 160 deg; joints [-0.927, 72.81, -12.214, -158.353, 62.354, 169.566]
  Call Extruder(1503.73388)
  MoveL 3063 to (519.98, 444.2, 52) mm, rotated rx -180 ry 0 rz 160 deg; joints [-0.835, 73.148, -12.967, -158.17, 61.985, 169.344]
  Call Extruder(1510.64393)
  MoveL 3064 to (522, 444.96, 52) mm, rotated rx -180 ry 0 rz 160 deg; joints [-0.739, 73.472, -13.688, -157.983, 61.635, 169.125]
  Set speed (17.6 mm/s)
  Call Extruder(1517.71880)
  MoveL 3065 to (524.03, 445.82, 52) mm, rotated rx -180 ry 0 rz 160 deg; joints [-0.632, 73.804, -14.423, -157.781, 61.282, 168.895]
  Set speed (17.6 mm/s)
  Call Extruder(1524.71676)
  MoveL 3066 to (526.01, 446.74, 52) mm, rotated rx -180 ry 0 rz 160 deg; joints [-0.518, 74.132, -15.147, -157.571, 60.938, 168.662]
  Set speed (17.6 mm/s)
  Call Extruder(1531.61486)
  MoveL 3067 to (527.93, 447.72, 52) mm, rotated rx 180 ry 0 rz 160 deg; joints [-0.398, 74.454, -15.855, -157.353, 60.605, 168.427]
  Set speed (17.6 mm/s)
  Call Extruder(1538.69617)
  MoveL 3068 to (529.86, 448.8, 52) mm, rotated rx 180 ry 0 rz 160 deg; joints [-0.268, 74.782, -16.576, -157.12, 60.269, 168.18]
  Set speed (17.6 mm/s)
  Call Extruder(1545.59735)
  MoveL 3069 to (531.7, 449.92, 52) mm, rotated rx -180 ry 0 rz 160 deg; joints [-0.134, 75.101, -17.273, -156.884, 59.948, 167.934]
  Set speed (17.6 mm/s)
  Call Extruder(1552.68479)
  MoveL 3070 to (533.54, 451.14, 52) mm, rotated rx 180 ry 0 rz 160 deg; joints [0.011, 75.425, -17.981, -156.632, 59.627, 167.676]
  Set speed (17.6 mm/s)
  Call Extruder(1559.52816)
  MoveL 3071 to (535.28, 452.38, 52) mm, rotated rx -180 ry 0 rz 160 deg; joints [0.158, 75.735, -18.656, -156.38, 59.324, 167.423]
  Set speed (17.6 mm/s)
  Call Extruder(1566.41873)
  MoveL 3072 to (536.99, 453.69, 52) mm, rotated rx -180 ry 0 rz 160 deg; joints [0.312, 76.044, -19.326, -156.118, 59.027, 167.164]
  Set speed (17.6 mm/s)
  Call Extruder(1573.41686)
  MoveL 3073 to (538.67, 455.08, 52) mm, rotated rx -180 ry 0 rz 160 deg; joints [0.475, 76.353, -19.996, -155.844, 58.734, 166.896]
  Call Extruder(0.00000)
  Set speed (17.6 mm/s)
  Call Extruder(7.13738)
  MoveL 3074 to (540.33, 456.57, 52) mm, rotated rx -180 ry 0 rz 160 deg; joints [0.647, 76.664, -20.667, -155.557, 58.444, 166.62]
  Set speed (17.6 mm/s)
  Call Extruder(14.19964)
  MoveL 3075 to (541.92, 458.1, 52) mm, rotated rx 180 ry 0 rz 160 deg; joints [0.823, 76.966, -21.318, -155.266, 58.168, 166.344]
  Set speed (17.6 mm/s)
  Call Extruder(17.99250)
  MoveL 3076 to (542.74, 458.94, 52) mm, rotated rx -180 ry 0 rz 160 deg; joints [0.92, 77.126, -21.662, -155.107, 58.025, 166.194]
  Set speed (17.6 mm/s)
  Call Extruder(21.81484)
  MoveL 3077 to (543.56, 459.81, 52) mm, rotated rx 180 ry 0 rz 160 deg; joints [1.019, 77.285, -22.004, -154.944, 57.883, 166.042]
  Call Extruder(25.77860)
  MoveL 3078 to (544.39, 460.73, 52) mm, rotated rx -180 ry 0 rz 160 deg; joints [1.124, 77.448, -22.354, -154.774, 57.739, 165.884]
  Set speed (17.6 mm/s)
  Call Extruder(29.71104)
  MoveL 3079 to (545.2, 461.66, 52) mm, rotated rx -180 ry 0 rz 160 deg; joints [1.23, 77.608, -22.696, -154.604, 57.6, 165.727]
  Set speed (17.6 mm/s)
  Call Extruder(33.52817)
  MoveL 3080 to (545.96, 462.57, 52) mm, rotated rx 180 ry 0 rz 160 deg; joints [1.334, 77.76, -23.023, -154.437, 57.468, 165.574]
  Set speed (17.6 mm/s)
  Call Extruder(38.17527)
  MoveL 3081 to (546.86, 463.71, 52) mm, rotated rx -180 ry 0 rz 160 deg; joints [1.463, 77.943, -23.414, -154.231, 57.313, 165.388]
  Set speed (17.6 mm/s)
  Call Extruder(41.42433)
  MoveL 3082 to (547.47, 464.52, 52) mm, rotated rx -180 ry 0 rz 160 deg; joints [1.554, 78.069, -23.683, -154.086, 57.207, 165.257]
  Set speed (17.6 mm/s)
  Call Extruder(44.68110)
  MoveL 3083 to (548.07, 465.34, 52) mm, rotated rx 180 ry 0 rz 160 deg; joints [1.646, 78.194, -23.949, -153.94, 57.104, 165.125]
  Set speed (17.6 mm/s)
  Call Extruder(49.09986)
  MoveL 3084 to (548.87, 466.46, 52) mm, rotated rx 180 ry 0 rz 160 deg; joints [1.773, 78.36, -24.303, -153.74, 56.968, 164.947]
  Set speed (17.6 mm/s)
  Call Extruder(52.98404)
  MoveL 3085 to (549.54, 467.47, 52) mm, rotated rx 180 ry 0 rz 160 deg; joints [1.886, 78.503, -24.607, -153.563, 56.853, 164.791]
  Set speed (17.6 mm/s)
  Call Extruder(56.77928)
  MoveL 3086 to (550.18, 468.47, 52) mm, rotated rx -180 ry 0 rz 160 deg; joints [1.998, 78.64, -24.899, -153.389, 56.744, 164.638]
  Set speed (17.6 mm/s)
  Call Extruder(60.67975)
  MoveL 3087 to (550.82, 469.5, 52) mm, rotated rx -180 ry 0 rz 160 deg; joints [2.114, 78.777, -25.191, -153.209, 56.637, 164.481]
  Set speed (17.6 mm/s)
  Call Extruder(64.64606)
  MoveL 3088 to (551.44, 470.57, 52) mm, rotated rx 180 ry 0 rz 160 deg; joints [2.233, 78.914, -25.482, -153.026, 56.532, 164.322]
  Set speed (17.6 mm/s)
  Call Extruder(69.64968)
  MoveL 3089 to (552.2, 471.93, 52) mm, rotated rx 180 ry 0 rz 160 deg; joints [2.385, 79.083, -25.84, -152.793, 56.405, 164.121]
  Set speed (17.6 mm/s)
  Call Extruder(72.34043)
  MoveL 3090 to (552.59, 472.68, 52) mm, rotated rx -180 ry 0 rz 160 deg; joints [2.468, 79.171, -26.026, -152.668, 56.34, 164.014]
  Set speed (17.6 mm/s)
  Call Extruder(76.20006)
  MoveL 3091 to (553.14, 473.75, 52) mm, rotated rx 180 ry 0 rz 160 deg; joints [2.588, 79.295, -26.289, -152.487, 56.25, 163.861]
  Call Extruder(80.27647)
  MoveL 3092 to (553.69, 474.9, 52) mm, rotated rx -180 ry 0 rz 160 deg; joints [2.715, 79.422, -26.558, -152.295, 56.16, 163.7]
  Set speed (17.6 mm/s)
  Call Extruder(84.05037)
  MoveL 3093 to (554.18, 475.97, 52) mm, rotated rx -180 ry 0 rz 160 deg; joints [2.834, 79.537, -26.8, -152.118, 56.08, 163.551]
  Call Extruder(91.71724)
  MoveL 3094 to (555.11, 478.18, 52) mm, rotated rx 180 ry 0 rz 160 deg; joints [3.079, 79.759, -27.269, -151.757, 55.932, 163.253]
  Set speed (17.6 mm/s)
  Call Extruder(95.72629)
  MoveL 3095 to (555.55, 479.34, 52) mm, rotated rx 180 ry 0 rz 160 deg; joints [3.209, 79.868, -27.499, -151.568, 55.864, 163.1]
  Set speed (17.6 mm/s)
  Call Extruder(99.55598)
  MoveL 3096 to (555.96, 480.46, 52) mm, rotated rx -180 ry 0 rz 160 deg; joints [3.333, 79.97, -27.715, -151.388, 55.8, 162.954]
  Set speed (17.6 mm/s)
  Call Extruder(103.50457)
  MoveL 3097 to (556.34, 481.63, 52) mm, rotated rx -180 ry 0 rz 160 deg; joints [3.462, 80.07, -27.924, -151.202, 55.742, 162.806]
  Set speed (17.6 mm/s)
  Call Extruder(107.54014)
  MoveL 3098 to (556.73, 482.83, 52) mm, rotated rx -180 ry 0 rz 160 deg; joints [3.595, 80.17, -28.134, -151.013, 55.685, 162.655]
  Set speed (17.6 mm/s)
  Call Extruder(115.06274)
  MoveL 3099 to (557.36, 485.09, 52) mm, rotated rx 180 ry 0 rz 160 deg; joints [3.845, 80.341, -28.496, -150.661, 55.594, 162.38]
  Set speed (17.6 mm/s)
  Call Extruder(122.82105)
  MoveL 3100 to (557.92, 487.45, 52) mm, rotated rx -180 ry 0 rz 160 deg; joints [4.105, 80.502, -28.833, -150.3, 55.52, 162.104]
  Set speed (17.6 mm/s)
  Call Extruder(130.67352)
  MoveL 3101 to (558.39, 489.85, 52) mm, rotated rx -180 ry 0 rz 160 deg; joints [4.372, 80.646, -29.135, -149.939, 55.465, 161.835]
  Set speed (17.6 mm/s)
  Call Extruder(138.44267)
  MoveL 3102 to (558.76, 492.25, 52) mm, rotated rx 180 ry 0 rz 160 deg; joints [4.637, 80.771, -29.396, -149.585, 55.431, 161.578]
  Set speed (17.6 mm/s)
  Call Extruder(146.30712)
  MoveL 3103 to (559.03, 494.69, 52) mm, rotated rx -180 ry 0 rz 160 deg; joints [4.908, 80.878, -29.62, -149.233, 55.416, 161.328]
  Set speed (17.6 mm/s)
  Call Extruder(153.97028)
  MoveL 3104 to (559.2, 497.08, 52) mm, rotated rx 180 ry 0 rz 160 deg; joints [5.173, 80.963, -29.798, -148.895, 55.421, 161.097]
  Set speed (17.6 mm/s)
  Call Extruder(161.74353)
  MoveL 3105 to (559.27, 499.5, 52) mm, rotated rx -180 ry 0 rz 160 deg; joints [5.443, 81.03, -29.939, -148.558, 55.447, 160.875]
  Set speed (17.6 mm/s)
  Call Extruder(169.38123)
  MoveL 3106 to (559.24, 501.89, 52) mm, rotated rx 180 ry 0 rz 160 deg; joints [5.71, 81.076, -30.037, -148.234, 55.491, 160.669]
  Set speed (17.6 mm/s)
  Call Extruder(177.26126)
  MoveL 3107 to (559.11, 504.34, 52) mm, rotated rx -180 ry 0 rz 160 deg; joints [5.985, 81.104, -30.095, -147.908, 55.557, 160.471]
  Set speed (17.6 mm/s)
  Call Extruder(184.95145)
  MoveL 3108 to (558.88, 506.73, 52) mm, rotated rx -180 ry 0 rz 160 deg; joints [6.254, 81.111, -30.11, -147.598, 55.641, 160.293]
  Set speed (17.6 mm/s)
  Call Extruder(192.90696)
  MoveL 3109 to (558.55, 509.19, 52) mm, rotated rx 180 ry 0 rz 160 deg; joints [6.532, 81.098, -30.082, -147.287, 55.747, 160.124]
  Set speed (17.6 mm/s)
  Call Extruder(200.57321)
  MoveL 3110 to (558.13, 511.55, 52) mm, rotated rx -180 ry 0 rz 160 deg; joints [6.8, 81.066, -30.015, -146.995, 55.868, 159.976]
  Set speed (17.6 mm/s)
  Call Extruder(208.38381)
  MoveL 3111 to (557.61, 513.93, 52) mm, rotated rx -180 ry 0 rz 160 deg; joints [7.072, 81.013, -29.903, -146.708, 56.01, 159.841]
  Set speed (17.6 mm/s)
  Call Extruder(216.11654)
  MoveL 3112 to (557, 516.26, 52) mm, rotated rx -180 ry 0 rz 160 deg; joints [7.341, 80.941, -29.752, -146.434, 56.169, 159.724]
  Call Extruder(223.76636)
  MoveL 3113 to (556.29, 518.55, 52) mm, rotated rx 180 ry 0 rz 160 deg; joints [7.605, 80.85, -29.563, -146.173, 56.343, 159.625]
  Call Extruder(231.53385)
  MoveL 3114 to (555.49, 520.83, 52) mm, rotated rx 180 ry 0 rz 160 deg; joints [7.872, 80.739, -29.33, -145.918, 56.537, 159.541]
  Set speed (17.6 mm/s)
  Call Extruder(235.55498)
  MoveL 3115 to (555.03, 522, 52) mm, rotated rx 180 ry 0 rz 160 deg; joints [8.009, 80.673, -29.192, -145.79, 56.644, 159.504]
  Set speed (17.6 mm/s)
  Call Extruder(239.55206)
  MoveL 3116 to (554.56, 523.15, 52) mm, rotated rx 180 ry 0 rz 160 deg; joints [8.145, 80.605, -29.05, -145.666, 56.754, 159.471]
  Set speed (17.6 mm/s)
  Call Extruder(247.03129)
  MoveL 3117 to (553.6, 525.28, 52) mm, rotated rx 180 ry 0 rz 160 deg; joints [8.398, 80.463, -28.751, -145.441, 56.972, 159.422]
  Set speed (17.6 mm/s)
  Call Extruder(251.00229)
  MoveL 3118 to (553.06, 526.4, 52) mm, rotated rx -180 ry 0 rz 160 deg; joints [8.531, 80.381, -28.578, -145.325, 57.093, 159.402]
  Set speed (17.6 mm/s)
  Call Extruder(254.97502)
  MoveL 3119 to (552.5, 527.51, 52) mm, rotated rx 180 ry 0 rz 160 deg; joints [8.664, 80.295, -28.398, -145.212, 57.218, 159.386]
  Set speed (17.6 mm/s)
  Call Extruder(258.80055)
  MoveL 3120 to (551.94, 528.56, 52) mm, rotated rx 180 ry 0 rz 160 deg; joints [8.791, 80.206, -28.212, -145.106, 57.342, 159.376]
  Set speed (17.6 mm/s)
  Call Extruder(262.64217)
  MoveL 3121 to (551.35, 529.6, 52) mm, rotated rx -180 ry 0 rz 160 deg; joints [8.918, 80.115, -28.019, -145.002, 57.47, 159.369]
  Set speed (17.6 mm/s)
  Call Extruder(266.55441)
  MoveL 3122 to (550.73, 530.65, 52) mm, rotated rx 180 ry 0 rz 160 deg; joints [9.047, 80.016, -27.812, -144.9, 57.604, 159.366]
  Set speed (17.6 mm/s)
  Call Extruder(270.41709)
  MoveL 3123 to (550.09, 531.68, 52) mm, rotated rx -180 ry 0 rz 160 deg; joints [9.173, 79.916, -27.6, -144.801, 57.74, 159.367]
  Set speed (17.6 mm/s)
  Call Extruder(273.65591)
  MoveL 3124 to (549.55, 532.53, 52) mm, rotated rx 180 ry 0 rz 160 deg; joints [9.278, 79.829, -27.416, -144.719, 57.855, 159.371]
  Set speed (17.6 mm/s)
  Call Extruder(278.21742)
  MoveL 3125 to (548.75, 533.71, 52) mm, rotated rx 180 ry 0 rz 160 deg; joints [9.425, 79.701, -27.146, -144.609, 58.023, 159.382]
  Set speed (17.6 mm/s)
  Call Extruder(282.07025)
  MoveL 3126 to (548.05, 534.69, 52) mm, rotated rx 180 ry 0 rz 160 deg; joints [9.547, 79.589, -26.91, -144.518, 58.168, 159.395]
  Call Extruder(285.97038)
  MoveL 3127 to (547.33, 535.67, 52) mm, rotated rx 180 ry 0 rz 160 deg; joints [9.671, 79.472, -26.664, -144.429, 58.317, 159.413]
  Set speed (17.6 mm/s)
  Call Extruder(289.82530)
  MoveL 3128 to (546.6, 536.62, 52) mm, rotated rx -180 ry 0 rz 160 deg; joints [9.792, 79.353, -26.412, -144.343, 58.467, 159.433]
  Set speed (17.6 mm/s)
  Call Extruder(293.73088)
  MoveL 3129 to (545.84, 537.58, 52) mm, rotated rx 180 ry 0 rz 160 deg; joints [9.914, 79.23, -26.15, -144.259, 58.622, 159.458]
  Set speed (17.6 mm/s)
  Call Extruder(297.66858)
  MoveL 3130 to (545.05, 538.52, 52) mm, rotated rx 180 ry 0 rz 160 deg; joints [10.035, 79.101, -25.878, -144.177, 58.781, 159.488]
  Set speed (17.6 mm/s)
  Call Extruder(301.57567)
  MoveL 3131 to (544.25, 539.44, 52) mm, rotated rx -180 ry 0 rz 160 deg; joints [10.154, 78.971, -25.602, -144.098, 58.941, 159.52]
  Set speed (17.6 mm/s)
  Call Extruder(305.38614)
  MoveL 3132 to (543.44, 540.32, 52) mm, rotated rx -180 ry 0 rz 160 deg; joints [10.27, 78.84, -25.325, -144.024, 59.1, 159.555]
  Set speed (17.6 mm/s)
  Call Extruder(308.57221)
  MoveL 3133 to (542.77, 541.04, 52) mm, rotated rx 180 ry 0 rz 160 deg; joints [10.365, 78.73, -25.09, -143.963, 59.234, 159.587]
  Set speed (17.6 mm/s)
  Call Extruder(313.14884)
  MoveL 3134 to (541.76, 542.06, 52) mm, rotated rx 180 ry 0 rz 160 deg; joints [10.501, 78.566, -24.743, -143.88, 59.43, 159.638]
  Set speed (17.6 mm/s)
  Call Extruder(317.04384)
  MoveL 3135 to (540.89, 542.91, 52) mm, rotated rx 180 ry 0 rz 160 deg; joints [10.615, 78.424, -24.44, -143.812, 59.599, 159.685]
  Set speed (17.6 mm/s)
  Call Extruder(320.93342)
  MoveL 3136 to (540, 543.73, 52) mm, rotated rx -180 ry 0 rz 160 deg; joints [10.727, 78.279, -24.131, -143.746, 59.77, 159.735]
  Set speed (17.6 mm/s)
  Call Extruder(324.80228)
  MoveL 3137 to (539.1, 544.54, 52) mm, rotated rx 180 ry 0 rz 160 deg; joints [10.837, 78.132, -23.818, -143.683, 59.943, 159.789]
  Set speed (17.6 mm/s)
  Call Extruder(328.72634)
  MoveL 3138 to (538.18, 545.34, 52) mm, rotated rx 180 ry 0 rz 160 deg; joints [10.948, 77.981, -23.496, -143.622, 60.119, 159.846]
  Set speed (17.6 mm/s)
  Call Extruder(332.68592)
  MoveL 3139 to (537.22, 546.12, 52) mm, rotated rx 180 ry 0 rz 160 deg; joints [11.058, 77.826, -23.164, -143.563, 60.298, 159.908]
  Set speed (17.6 mm/s)
  Call Extruder(337.25700)
  MoveL 3140 to (536.1, 547, 52) mm, rotated rx -180 ry 0 rz 160 deg; joints [11.183, 77.644, -22.775, -143.498, 60.508, 159.983]
  Call Extruder(340.34935)
  MoveL 3141 to (535.33, 547.58, 52) mm, rotated rx -180 ry 0 rz 160 deg; joints [11.267, 77.519, -22.507, -143.456, 60.651, 160.036]
  Set speed (17.6 mm/s)
  Call Extruder(344.26266)
  MoveL 3142 to (534.35, 548.3, 52) mm, rotated rx -180 ry 0 rz 160 deg; joints [11.371, 77.36, -22.164, -143.404, 60.834, 160.106]
  Set speed (17.6 mm/s)
  Call Extruder(348.12727)
  MoveL 3143 to (533.36, 548.99, 52) mm, rotated rx 180 ry 0 rz 160 deg; joints [11.472, 77.2, -21.821, -143.356, 61.016, 160.178]
  Call Extruder(352.13329)
  MoveL 3144 to (532.32, 549.69, 52) mm, rotated rx 180 ry 0 rz 160 deg; joints [11.576, 77.032, -21.46, -143.309, 61.205, 160.256]
  Set speed (17.6 mm/s)
  Call Extruder(355.77049)
  MoveL 3145 to (531.36, 550.29, 52) mm, rotated rx 180 ry 0 rz 160 deg; joints [11.667, 76.877, -21.127, -143.269, 61.379, 160.33]
  Set speed (17.6 mm/s)
  Call Extruder(359.79723)
  MoveL 3146 to (530.28, 550.95, 52) mm, rotated rx -180 ry 0 rz 160 deg; joints [11.768, 76.705, -20.756, -143.226, 61.572, 160.414]
  Set speed (17.6 mm/s)
  Call Extruder(363.65781)
  MoveL 3147 to (529.24, 551.55, 52) mm, rotated rx -180 ry 0 rz 160 deg; joints [11.862, 76.538, -20.396, -143.187, 61.759, 160.498]
  Set speed (17.6 mm/s)
  Call Extruder(366.97468)
  MoveL 3148 to (528.34, 552.06, 52) mm, rotated rx 180 ry 0 rz 160 deg; joints [11.942, 76.394, -20.084, -143.156, 61.92, 160.572]
  Set speed (17.6 mm/s)
  Call Extruder(372.56775)
  MoveL 3149 to (526.79, 552.87, 52) mm, rotated rx 180 ry 0 rz 160 deg; joints [12.073, 76.147, -19.55, -143.107, 62.192, 160.701]
  Set speed (17.6 mm/s)
  Call Extruder(375.36355)
  MoveL 3150 to (526.01, 553.26, 52) mm, rotated rx 180 ry 0 rz 160 deg; joints [12.137, 76.023, -19.281, -143.085, 62.33, 160.768]
  Set speed (17.6 mm/s)
  Call Extruder(379.19007)
  MoveL 3151 to (524.94, 553.77, 52) mm, rotated rx -180 ry 0 rz 160 deg; joints [12.223, 75.852, -18.91, -143.056, 62.518, 160.861]
  Set speed (17.6 mm/s)
  Call Extruder(383.19892)
  MoveL 3152 to (523.79, 554.28, 52) mm, rotated rx -180 ry 0 rz 160 deg; joints [12.31, 75.671, -18.517, -143.029, 62.716, 160.962]
  Set speed (17.6 mm/s)
  Call Extruder(386.96790)
  MoveL 3153 to (522.72, 554.74, 52) mm, rotated rx 180 ry 0 rz 160 deg; joints [12.391, 75.501, -18.147, -143.005, 62.902, 161.058]
  Set speed (17.6 mm/s)
  Call Extruder(390.95414)
  MoveL 3154 to (521.56, 555.2, 52) mm, rotated rx 180 ry 0 rz 160 deg; joints [12.474, 75.32, -17.751, -142.983, 63.1, 161.163]
  Set speed (17.6 mm/s)
  Call Extruder(394.75193)
  MoveL 3155 to (520.46, 555.63, 52) mm, rotated rx -180 ry 0 rz 160 deg; joints [12.552, 75.146, -17.373, -142.962, 63.289, 161.264]
  Call Extruder(398.78972)
  MoveL 3156 to (519.27, 556.04, 52) mm, rotated rx -180 ry 0 rz 160 deg; joints [12.631, 74.96, -16.966, -142.945, 63.491, 161.375]
  Set speed (17.6 mm/s)
  Call Extruder(402.51914)
  MoveL 3157 to (518.17, 556.41, 52) mm, rotated rx -180 ry 0 rz 160 deg; joints [12.703, 74.789, -16.59, -142.93, 63.676, 161.479]
  Set speed (17.6 mm/s)
  Call Extruder(406.52447)
  MoveL 3158 to (516.98, 556.78, 52) mm, rotated rx -180 ry 0 rz 160 deg; joints [12.777, 74.603, -16.183, -142.917, 63.877, 161.593]
  Set speed (17.6 mm/s)
  Call Extruder(410.24859)
  MoveL 3159 to (515.86, 557.11, 52) mm, rotated rx -180 ry 0 rz 160 deg; joints [12.845, 74.43, -15.803, -142.906, 64.063, 161.7]
  Call Extruder(413.76702)
  MoveL 3160 to (514.8, 557.39, 52) mm, rotated rx 180 ry 0 rz 160 deg; joints [12.906, 74.266, -15.443, -142.899, 64.239, 161.804]
  Set speed (17.6 mm/s)
  Call Extruder(418.03998)
  MoveL 3161 to (513.51, 557.71, 52) mm, rotated rx 180 ry 0 rz 160 deg; joints [12.979, 74.067, -15.004, -142.892, 64.453, 161.931]
  Set speed (17.6 mm/s)
  Call Extruder(425.95045)
  MoveL 3162 to (511.1, 558.22, 52) mm, rotated rx 180 ry 0 rz 160 deg; joints [13.105, 73.697, -14.185, -142.887, 64.849, 162.174]
  Set speed (17.6 mm/s)
  Call Extruder(433.78043)
  MoveL 3163 to (508.69, 558.63, 52) mm, rotated rx 180 ry 0 rz 160 deg; joints [13.22, 73.329, -13.37, -142.892, 65.241, 162.421]
  Set speed (17.6 mm/s)
  Call Extruder(441.47523)
  MoveL 3164 to (506.3, 558.93, 52) mm, rotated rx 180 ry 0 rz 160 deg; joints [13.323, 72.968, -12.566, -142.906, 65.625, 162.669]
  Set speed (17.6 mm/s)
  Call Extruder(449.27722)
  MoveL 3165 to (503.88, 559.14, 52) mm, rotated rx 180 ry 0 rz 160 deg; joints [13.417, 72.602, -11.749, -142.93, 66.013, 162.927]
  Set speed (17.6 mm/s)
  Call Extruder(457.08526)
  MoveL 3166 to (501.44, 559.25, 52) mm, rotated rx 180 ry 0 rz 160 deg; joints [13.5, 72.237, -10.93, -142.964, 66.399, 163.191]
  Set speed (17.6 mm/s)
  Call Extruder(464.75929)
  MoveL 3167 to (499.05, 559.26, 52) mm, rotated rx 180 ry 0 rz 160 deg; joints [13.571, 71.88, -10.127, -143.006, 66.775, 163.454]
  Set speed (10.0 mm/s)
  MoveL 3168 to (499.05, 559.26, 56) mm, rotated rx -180 ry 0 rz 160 deg; joints [13.571, 71.188, -9.69, -142.94, 66.572, 163.287]
  Set speed (120.0 mm/s)
  MoveL 3169 to (499.03, 560.1, 56) mm, rotated rx -180 ry 0 rz 160 deg; joints [13.672, 71.216, -9.752, -142.826, 66.574, 163.223]
  Set speed (17.6 mm/s)
  Call Extruder(472.54096)
  MoveL 3170 to (501.46, 560.09, 56) mm, rotated rx 180 ry 0 rz 160 deg; joints [13.6, 71.579, -10.565, -142.782, 66.195, 162.956]
  Set speed (17.6 mm/s)
  Call Extruder(480.46032)
  MoveL 3171 to (503.93, 559.97, 56) mm, rotated rx 180 ry 0 rz 160 deg; joints [13.515, 71.951, -11.394, -142.748, 65.806, 162.69]
  Call Extruder(488.12747)
  MoveL 3172 to (506.32, 559.77, 56) mm, rotated rx -180 ry 0 rz 160 deg; joints [13.422, 72.312, -12.195, -142.724, 65.427, 162.437]
  Set speed (17.6 mm/s)
  Call Extruder(496.15219)
  MoveL 3173 to (508.81, 559.45, 56) mm, rotated rx -180 ry 0 rz 160 deg; joints [13.315, 72.69, -13.032, -142.709, 65.029, 162.178]
  Call Extruder(504.07617)
  MoveL 3174 to (511.25, 559.04, 56) mm, rotated rx 180 ry 0 rz 160 deg; joints [13.198, 73.063, -13.856, -142.703, 64.635, 161.928]
  Set speed (17.6 mm/s)
  Call Extruder(511.75613)
  MoveL 3175 to (513.6, 558.54, 56) mm, rotated rx -180 ry 0 rz 160 deg; joints [13.075, 73.424, -14.649, -142.707, 64.253, 161.694]
  Set speed (17.6 mm/s)
  Call Extruder(516.43753)
  MoveL 3176 to (515.02, 558.19, 56) mm, rotated rx -180 ry 0 rz 160 deg; joints [12.995, 73.643, -15.13, -142.715, 64.02, 161.554]
  Call Extruder(519.63067)
  MoveL 3177 to (515.98, 557.94, 56) mm, rotated rx -180 ry 0 rz 160 deg; joints [12.94, 73.792, -15.457, -142.72, 63.86, 161.46]
  Set speed (17.6 mm/s)
  Call Extruder(523.77271)
  MoveL 3178 to (517.22, 557.58, 56) mm, rotated rx -180 ry 0 rz 160 deg; joints [12.864, 73.985, -15.878, -142.732, 63.654, 161.341]
  Call Extruder(527.55875)
  MoveL 3179 to (518.35, 557.24, 56) mm, rotated rx 180 ry 0 rz 160 deg; joints [12.794, 74.161, -16.263, -142.743, 63.466, 161.233]
  Set speed (17.6 mm/s)
  Call Extruder(531.59116)
  MoveL 3180 to (519.54, 556.83, 56) mm, rotated rx -180 ry 0 rz 160 deg; joints [12.716, 74.347, -16.669, -142.76, 63.266, 161.121]
  Set speed (17.6 mm/s)
  Call Extruder(535.45243)
  MoveL 3181 to (520.68, 556.43, 56) mm, rotated rx 180 ry 0 rz 160 deg; joints [12.64, 74.526, -17.057, -142.776, 63.074, 161.015]
  Call Extruder(539.50983)
  MoveL 3182 to (521.86, 555.98, 56) mm, rotated rx -180 ry 0 rz 160 deg; joints [12.557, 74.711, -17.46, -142.797, 62.873, 160.908]
  Set speed (17.6 mm/s)
  Call Extruder(543.22788)
  MoveL 3183 to (522.94, 555.55, 56) mm, rotated rx -180 ry 0 rz 160 deg; joints [12.479, 74.881, -17.83, -142.817, 62.689, 160.81]
  Call Extruder(547.38875)
  MoveL 3184 to (524.14, 555.04, 56) mm, rotated rx 180 ry 0 rz 160 deg; joints [12.39, 75.07, -18.238, -142.843, 62.485, 160.704]
  Set speed (17.6 mm/s)
  Call Extruder(551.19157)
  MoveL 3185 to (525.22, 554.56, 56) mm, rotated rx -180 ry 0 rz 160 deg; joints [12.306, 75.241, -18.61, -142.869, 62.298, 160.609]
  Set speed (17.6 mm/s)
  Call Extruder(555.13262)
  MoveL 3186 to (526.33, 554.03, 56) mm, rotated rx 180 ry 0 rz 160 deg; joints [12.218, 75.418, -18.992, -142.898, 62.105, 160.513]
  Set speed (17.7 mm/s)
  Call Extruder(561.06092)
  MoveL 3187 to (527.99, 553.2, 56) mm, rotated rx 180 ry 0 rz 160 deg; joints [12.081, 75.683, -19.562, -142.946, 61.815, 160.373]
  Call Extruder(567.04230)
  MoveL 3188 to (529.63, 552.29, 56) mm, rotated rx -180 ry 0 rz 160 deg; joints [11.938, 75.945, -20.127, -143.001, 61.525, 160.239]
  Set speed (17.6 mm/s)
  Call Extruder(570.91509)
  MoveL 3189 to (530.67, 551.69, 56) mm, rotated rx -180 ry 0 rz 160 deg; joints [11.843, 76.113, -20.487, -143.039, 61.339, 160.155]
  Call Extruder(574.84574)
  MoveL 3190 to (531.73, 551.05, 56) mm, rotated rx -180 ry 0 rz 160 deg; joints [11.745, 76.282, -20.85, -143.08, 61.151, 160.073]
  Set speed (17.6 mm/s)
  Call Extruder(578.78479)
  MoveL 3191 to (532.76, 550.39, 56) mm, rotated rx -180 ry 0 rz 160 deg; joints [11.645, 76.449, -21.209, -143.124, 60.963, 159.993]
  Call Extruder(582.67060)
  MoveL 3192 to (533.77, 549.72, 56) mm, rotated rx 180 ry 0 rz 160 deg; joints [11.545, 76.612, -21.559, -143.17, 60.78, 159.918]
  Set speed (17.6 mm/s)
  Call Extruder(586.57762)
  MoveL 3193 to (534.78, 549.02, 56) mm, rotated rx -180 ry 0 rz 160 deg; joints [11.443, 76.775, -21.906, -143.218, 60.597, 159.845]
  Set speed (17.6 mm/s)
  Call Extruder(590.60165)
  MoveL 3194 to (535.79, 548.28, 56) mm, rotated rx -180 ry 0 rz 160 deg; joints [11.335, 76.939, -22.258, -143.27, 60.41, 159.773]
  Call Extruder(594.44984)
  MoveL 3195 to (536.75, 547.56, 56) mm, rotated rx -180 ry 0 rz 160 deg; joints [11.231, 77.095, -22.59, -143.322, 60.232, 159.707]
  Set speed (17.6 mm/s)
  Call Extruder(598.45256)
  MoveL 3196 to (537.73, 546.78, 56) mm, rotated rx 180 ry 0 rz 160 deg; joints [11.122, 77.255, -22.931, -143.379, 60.049, 159.642]
  Call Extruder(602.38062)
  MoveL 3197 to (538.68, 546, 56) mm, rotated rx -180 ry 0 rz 160 deg; joints [11.012, 77.409, -23.259, -143.437, 59.871, 159.581]
  Set speed (17.6 mm/s)
  Call Extruder(606.32462)
  MoveL 3198 to (539.62, 545.2, 56) mm, rotated rx 180 ry 0 rz 160 deg; joints [10.901, 77.561, -23.583, -143.498, 59.694, 159.524]
  Call Extruder(610.20276)
  MoveL 3199 to (540.52, 544.39, 56) mm, rotated rx 180 ry 0 rz 160 deg; joints [10.79, 77.709, -23.897, -143.561, 59.522, 159.47]
  Call Extruder(614.19006)
  MoveL 3200 to (541.43, 543.54, 56) mm, rotated rx -180 ry 0 rz 160 deg; joints [10.675, 77.857, -24.212, -143.628, 59.347, 159.419]
  Set speed (17.6 mm/s)
  Call Extruder(618.20203)
  MoveL 3201 to (542.33, 542.67, 56) mm, rotated rx -180 ry 0 rz 160 deg; joints [10.557, 78.005, -24.524, -143.698, 59.173, 159.371]
  Set speed (17.6 mm/s)
  Call Extruder(622.05217)
  MoveL 3202 to (543.18, 541.81, 56) mm, rotated rx 180 ry 0 rz 160 deg; joints [10.443, 78.143, -24.816, -143.767, 59.009, 159.328]
  Set speed (17.6 mm/s)
  Call Extruder(625.98335)
  MoveL 3203 to (544.02, 540.92, 56) mm, rotated rx 180 ry 0 rz 160 deg; joints [10.326, 78.281, -25.109, -143.841, 58.842, 159.288]
  Set speed (17.6 mm/s)
  Call Extruder(629.93078)
  MoveL 3204 to (544.85, 540.01, 56) mm, rotated rx -180 ry 0 rz 160 deg; joints [10.206, 78.416, -25.395, -143.918, 58.678, 159.252]
  Call Extruder(633.84622)
  MoveL 3205 to (545.66, 539.09, 56) mm, rotated rx 180 ry 0 rz 160 deg; joints [10.087, 78.547, -25.672, -143.996, 58.518, 159.219]
  Call Extruder(637.79502)
  MoveL 3206 to (546.45, 538.14, 56) mm, rotated rx 180 ry 0 rz 160 deg; joints [9.965, 78.676, -25.944, -144.078, 58.359, 159.191]
  Call Extruder(641.71575)
  MoveL 3207 to (547.22, 537.19, 56) mm, rotated rx 180 ry 0 rz 160 deg; joints [9.843, 78.801, -26.207, -144.162, 58.203, 159.166]
  Set speed (17.6 mm/s)
  Call Extruder(645.58632)
  MoveL 3208 to (547.96, 536.23, 56) mm, rotated rx -180 ry 0 rz 160 deg; joints [9.721, 78.921, -26.46, -144.248, 58.052, 159.145]
  Call Extruder(649.59096)
  MoveL 3209 to (548.7, 535.22, 56) mm, rotated rx -180 ry 0 rz 160 deg; joints [9.595, 79.041, -26.714, -144.339, 57.899, 159.127]
  Set speed (17.6 mm/s)
  Call Extruder(653.51140)
  MoveL 3210 to (549.41, 534.22, 56) mm, rotated rx 180 ry 0 rz 160 deg; joints [9.47, 79.156, -26.954, -144.431, 57.752, 159.114]
  Set speed (17.6 mm/s)
  Call Extruder(658.20344)
  MoveL 3211 to (550.23, 533.01, 56) mm, rotated rx -180 ry 0 rz 160 deg; joints [9.319, 79.287, -27.231, -144.544, 57.58, 159.104]
  Call Extruder(661.39070)
  MoveL 3212 to (550.77, 532.17, 56) mm, rotated rx 180 ry 0 rz 160 deg; joints [9.215, 79.373, -27.411, -144.623, 57.466, 159.1]
  Set speed (17.6 mm/s)
  Call Extruder(665.31573)
  MoveL 3213 to (551.42, 531.13, 56) mm, rotated rx -180 ry 0 rz 160 deg; joints [9.087, 79.476, -27.626, -144.724, 57.328, 159.099]
  Call Extruder(669.25751)
  MoveL 3214 to (552.04, 530.07, 56) mm, rotated rx 180 ry 0 rz 160 deg; joints [8.958, 79.575, -27.834, -144.827, 57.194, 159.102]
  Set speed (17.6 mm/s)
  Call Extruder(673.18619)
  MoveL 3215 to (552.65, 529, 56) mm, rotated rx 180 ry 0 rz 160 deg; joints [8.828, 79.67, -28.033, -144.933, 57.062, 159.11]
  Set speed (17.6 mm/s)
  Call Extruder(677.12370)
  MoveL 3216 to (553.23, 527.91, 56) mm, rotated rx 180 ry 0 rz 160 deg; joints [8.697, 79.76, -28.222, -145.042, 56.934, 159.121]
  Set speed (17.6 mm/s)
  Call Extruder(682.34901)
  MoveL 3217 to (553.97, 526.46, 56) mm, rotated rx -180 ry 0 rz 160 deg; joints [8.523, 79.874, -28.461, -145.19, 56.77, 159.143]
  Set speed (17.6 mm/s)
  Call Extruder(685.17227)
  MoveL 3218 to (554.35, 525.67, 56) mm, rotated rx 180 ry 0 rz 160 deg; joints [8.428, 79.931, -28.581, -145.272, 56.685, 159.158]
  Set speed (17.6 mm/s)
  Call Extruder(692.84330)
  MoveL 3219 to (555.33, 523.48, 56) mm, rotated rx 180 ry 0 rz 160 deg; joints [8.169, 80.078, -28.888, -145.503, 56.461, 159.209]
  Set speed (17.6 mm/s)
  Call Extruder(696.88922)
  MoveL 3220 to (555.8, 522.31, 56) mm, rotated rx 180 ry 0 rz 160 deg; joints [8.031, 80.147, -29.031, -145.629, 56.35, 159.243]
  Call Extruder(700.71260)
  MoveL 3221 to (556.24, 521.2, 56) mm, rotated rx 180 ry 0 rz 160 deg; joints [7.901, 80.21, -29.163, -145.75, 56.247, 159.278]
  Set speed (17.6 mm/s)
  Call Extruder(708.62333)
  MoveL 3222 to (557.07, 518.87, 56) mm, rotated rx 180 ry 0 rz 160 deg; joints [7.629, 80.323, -29.4, -146.009, 56.049, 159.365]
  Set speed (17.6 mm/s)
  Call Extruder(712.61752)
  MoveL 3223 to (557.44, 517.68, 56) mm, rotated rx -180 ry 0 rz 160 deg; joints [7.492, 80.372, -29.501, -146.145, 55.957, 159.417]
  Set speed (17.6 mm/s)
  Call Extruder(716.41433)
  MoveL 3224 to (557.78, 516.54, 56) mm, rotated rx 180 ry 0 rz 160 deg; joints [7.36, 80.416, -29.593, -146.275, 55.871, 159.468]
  Call Extruder(720.51729)
  MoveL 3225 to (558.12, 515.31, 56) mm, rotated rx -180 ry 0 rz 160 deg; joints [7.218, 80.456, -29.676, -146.42, 55.785, 159.529]
  Set speed (17.6 mm/s)
  Call Extruder(724.41771)
  MoveL 3226 to (558.42, 514.13, 56) mm, rotated rx -180 ry 0 rz 160 deg; joints [7.083, 80.491, -29.751, -146.559, 55.706, 159.59]
  Set speed (17.6 mm/s)
  Call Extruder(732.32951)
  MoveL 3227 to (558.95, 511.71, 56) mm, rotated rx 180 ry 0 rz 160 deg; joints [6.807, 80.545, -29.863, -146.85, 55.561, 159.727]
  Set speed (17.6 mm/s)
  Call Extruder(740.02938)
  MoveL 3228 to (559.37, 509.34, 56) mm, rotated rx 180 ry 0 rz 160 deg; joints [6.538, 80.578, -29.931, -147.143, 55.439, 159.878]
  Call Extruder(747.81737)
  MoveL 3229 to (559.7, 506.93, 56) mm, rotated rx 180 ry 0 rz 160 deg; joints [6.266, 80.591, -29.959, -147.448, 55.333, 160.044]
  Set speed (17.6 mm/s)
  Call Extruder(755.92500)
  MoveL 3230 to (559.94, 504.41, 56) mm, rotated rx 180 ry 0 rz 160 deg; joints [5.983, 80.584, -29.945, -147.775, 55.243, 160.234]
  Set speed (17.6 mm/s)
  Call Extruder(763.58299)
  MoveL 3231 to (560.07, 502.02, 56) mm, rotated rx 180 ry 0 rz 160 deg; joints [5.715, 80.558, -29.889, -148.093, 55.178, 160.428]
  Set speed (17.6 mm/s)
  Call Extruder(771.66432)
  MoveL 3232 to (560.1, 499.49, 56) mm, rotated rx 180 ry 0 rz 160 deg; joints [5.433, 80.508, -29.786, -148.436, 55.129, 160.647]
  Set speed (17.6 mm/s)
  Call Extruder(779.53059)
  MoveL 3233 to (560.03, 497.04, 56) mm, rotated rx -180 ry 0 rz 160 deg; joints [5.16, 80.441, -29.645, -148.777, 55.102, 160.873]
  Call Extruder(787.23326)
  MoveL 3234 to (559.86, 494.63, 56) mm, rotated rx -180 ry 0 rz 160 deg; joints [4.894, 80.355, -29.466, -149.118, 55.095, 161.108]
  Set speed (17.6 mm/s)
  Call Extruder(795.26228)
  MoveL 3235 to (559.59, 492.14, 56) mm, rotated rx -180 ry 0 rz 160 deg; joints [4.617, 80.245, -29.238, -149.479, 55.108, 161.364]
  Set speed (17.6 mm/s)
  Call Extruder(803.13578)
  MoveL 3236 to (559.22, 489.71, 56) mm, rotated rx 180 ry 0 rz 160 deg; joints [4.349, 80.119, -28.973, -149.838, 55.142, 161.627]
  Set speed (17.6 mm/s)
  Call Extruder(811.04530)
  MoveL 3237 to (558.74, 487.29, 56) mm, rotated rx 180 ry 0 rz 160 deg; joints [4.081, 79.974, -28.669, -150.204, 55.196, 161.901]
  Set speed (17.6 mm/s)
  Call Extruder(814.91656)
  MoveL 3238 to (558.47, 486.11, 56) mm, rotated rx 180 ry 0 rz 160 deg; joints [3.951, 79.894, -28.504, -150.384, 55.231, 162.039]
  Set speed (17.6 mm/s)
  Call Extruder(818.82619)
  MoveL 3239 to (558.18, 484.92, 56) mm, rotated rx -180 ry 0 rz 160 deg; joints [3.82, 79.812, -28.332, -150.566, 55.268, 162.179]
  Set speed (17.6 mm/s)
  Call Extruder(822.81529)
  MoveL 3240 to (557.85, 483.72, 56) mm, rotated rx -180 ry 0 rz 160 deg; joints [3.687, 79.722, -28.143, -150.753, 55.314, 162.325]
  Set speed (17.6 mm/s)
  Call Extruder(826.49603)
  MoveL 3241 to (557.53, 482.62, 56) mm, rotated rx -180 ry 0 rz 160 deg; joints [3.565, 79.637, -27.965, -150.926, 55.358, 162.461]
  Set speed (17.6 mm/s)
  Call Extruder(830.67210)
  MoveL 3242 to (557.14, 481.38, 56) mm, rotated rx -180 ry 0 rz 160 deg; joints [3.428, 79.534, -27.749, -151.123, 55.416, 162.618]
  Set speed (17.6 mm/s)
  Call Extruder(834.52713)
  MoveL 3243 to (556.76, 480.24, 56) mm, rotated rx 180 ry 0 rz 160 deg; joints [3.302, 79.437, -27.546, -151.305, 55.472, 162.763]
  Call Extruder(838.57930)
  MoveL 3244 to (556.33, 479.05, 56) mm, rotated rx -180 ry 0 rz 160 deg; joints [3.17, 79.329, -27.318, -151.496, 55.538, 162.918]
  Set speed (17.6 mm/s)
  Call Extruder(842.92993)
  MoveL 3245 to (555.85, 477.78, 56) mm, rotated rx -180 ry 0 rz 160 deg; joints [3.03, 79.21, -27.068, -151.701, 55.612, 163.086]
  Set speed (17.6 mm/s)
  Call Extruder(850.22889)
  MoveL 3246 to (554.96, 475.68, 56) mm, rotated rx 180 ry 0 rz 160 deg; joints [2.797, 78.998, -26.622, -152.047, 55.751, 163.372]
  Set speed (17.6 mm/s)
  Call Extruder(854.18401)
  MoveL 3247 to (554.45, 474.56, 56) mm, rotated rx 180 ry 0 rz 160 deg; joints [2.673, 78.878, -26.369, -152.233, 55.833, 163.528]
  Call Extruder(858.16987)
  MoveL 3248 to (553.91, 473.43, 56) mm, rotated rx -180 ry 0 rz 160 deg; joints [2.548, 78.754, -26.107, -152.421, 55.92, 163.686]
  Call Extruder(862.07359)
  MoveL 3249 to (553.36, 472.34, 56) mm, rotated rx 180 ry 0 rz 160 deg; joints [2.427, 78.628, -25.843, -152.605, 56.009, 163.842]
  Set speed (17.6 mm/s)
  Call Extruder(866.05797)
  MoveL 3250 to (552.78, 471.25, 56) mm, rotated rx -180 ry 0 rz 160 deg; joints [2.304, 78.497, -25.565, -152.792, 56.105, 164.002]
  Call Extruder(869.96214)
  MoveL 3251 to (552.18, 470.18, 56) mm, rotated rx 180 ry 0 rz 160 deg; joints [2.185, 78.364, -25.286, -152.974, 56.204, 164.16]
  Set speed (17.6 mm/s)
  Call Extruder(873.86642)
  MoveL 3252 to (551.57, 469.13, 56) mm, rotated rx 180 ry 0 rz 160 deg; joints [2.068, 78.229, -24.999, -153.156, 56.306, 164.318]
  Set speed (17.6 mm/s)
  Call Extruder(877.83968)
  MoveL 3253 to (550.92, 468.07, 56) mm, rotated rx 180 ry 0 rz 160 deg; joints [1.949, 78.089, -24.702, -153.34, 56.415, 164.478]
  Set speed (17.6 mm/s)
  Call Extruder(881.84332)
  MoveL 3254 to (550.24, 467.02, 56) mm, rotated rx 180 ry 0 rz 160 deg; joints [1.831, 77.944, -24.395, -153.525, 56.528, 164.641]
  Set speed (17.6 mm/s)
  Call Extruder(885.70722)
  MoveL 3255 to (549.57, 466.01, 56) mm, rotated rx 180 ry 0 rz 160 deg; joints [1.719, 77.801, -24.092, -153.702, 56.642, 164.797]
  Set speed (17.6 mm/s)
  Call Extruder(889.63706)
  MoveL 3256 to (548.86, 465.01, 56) mm, rotated rx 180 ry 0 rz 160 deg; joints [1.606, 77.653, -23.779, -153.881, 56.761, 164.957]
  Set speed (17.6 mm/s)
  Call Extruder(893.66257)
  MoveL 3257 to (548.12, 463.99, 56) mm, rotated rx -180 ry 0 rz 160 deg; joints [1.491, 77.5, -23.452, -154.062, 56.887, 165.12]
  Set speed (17.6 mm/s)
  Call Extruder(897.49155)
  MoveL 3258 to (547.4, 463.04, 56) mm, rotated rx 180 ry 0 rz 160 deg; joints [1.384, 77.351, -23.135, -154.234, 57.011, 165.275]
  Set speed (17.6 mm/s)
  Call Extruder(901.45028)
  MoveL 3259 to (546.63, 462.07, 56) mm, rotated rx 180 ry 0 rz 160 deg; joints [1.274, 77.194, -22.802, -154.41, 57.142, 165.435]
  Set speed (17.6 mm/s)
  Call Extruder(905.36346)
  MoveL 3260 to (545.84, 461.13, 56) mm, rotated rx 180 ry 0 rz 160 deg; joints [1.167, 77.037, -22.467, -154.582, 57.276, 165.592]
  Set speed (17.6 mm/s)
  Call Extruder(909.46173)
  MoveL 3261 to (545.01, 460.17, 56) mm, rotated rx -180 ry 0 rz 160 deg; joints [1.057, 76.871, -22.111, -154.761, 57.42, 165.757]
  Set speed (17.6 mm/s)
  Call Extruder(913.23446)
  MoveL 3262 to (544.22, 459.29, 56) mm, rotated rx 180 ry 0 rz 160 deg; joints [0.957, 76.715, -21.779, -154.923, 57.556, 165.908]
  Set speed (17.6 mm/s)
  Call Extruder(917.19419)
  MoveL 3263 to (543.37, 458.39, 56) mm, rotated rx 180 ry 0 rz 160 deg; joints [0.854, 76.55, -21.425, -155.093, 57.701, 166.066]
  Set speed (17.6 mm/s)
  Call Extruder(921.03092)
  MoveL 3264 to (542.53, 457.53, 56) mm, rotated rx 180 ry 0 rz 160 deg; joints [0.756, 76.388, -21.078, -155.254, 57.846, 166.218]
  Set speed (17.6 mm/s)
  Call Extruder(928.20207)
  MoveL 3265 to (540.92, 455.98, 56) mm, rotated rx 180 ry 0 rz 160 deg; joints [0.576, 76.08, -20.418, -155.552, 58.124, 166.5]
  Set speed (17.6 mm/s)
  Call Extruder(935.16706)
  MoveL 3266 to (539.29, 454.52, 56) mm, rotated rx -180 ry 0 rz 160 deg; joints [0.408, 75.776, -19.764, -155.833, 58.404, 166.77]
  Call Extruder(942.24841)
  MoveL 3267 to (537.59, 453.11, 56) mm, rotated rx 180 ry 0 rz 160 deg; joints [0.243, 75.463, -19.088, -156.112, 58.698, 167.042]
  Set speed (17.6 mm/s)
  Call Extruder(949.36834)
  MoveL 3268 to (535.83, 451.75, 56) mm, rotated rx -180 ry 0 rz 160 deg; joints [0.083, 75.143, -18.396, -156.385, 59.002, 167.311]
  Set speed (17.6 mm/s)
  Call Extruder(956.36716)
  MoveL 3269 to (534.05, 450.48, 56) mm, rotated rx -180 ry 0 rz 160 deg; joints [-0.067, 74.825, -17.707, -156.644, 59.31, 167.571]
  Call Extruder(963.68177)
  MoveL 3270 to (532.14, 449.22, 56) mm, rotated rx -180 ry 0 rz 160 deg; joints [-0.218, 74.489, -16.978, -156.906, 59.64, 167.837]
  Call Extruder(970.66326)
  MoveL 3271 to (530.28, 448.08, 56) mm, rotated rx 180 ry 0 rz 160 deg; joints [-0.354, 74.166, -16.275, -157.147, 59.962, 168.087]
  Set speed (17.6 mm/s)
  Call Extruder(977.83810)
  MoveL 3272 to (528.32, 446.99, 56) mm, rotated rx -180 ry 0 rz 160 deg; joints [-0.486, 73.832, -15.544, -157.384, 60.3, 168.338]
  Set speed (17.6 mm/s)
  Call Extruder(984.72961)
  MoveL 3273 to (526.4, 446.01, 56) mm, rotated rx 180 ry 0 rz 160 deg; joints [-0.606, 73.51, -14.838, -157.603, 60.631, 168.573]
  Set speed (17.6 mm/s)
  Call Extruder(991.91113)
  MoveL 3274 to (524.37, 445.06, 56) mm, rotated rx 180 ry 0 rz 160 deg; joints [-0.724, 73.173, -14.097, -157.82, 60.981, 168.813]
  Set speed (17.6 mm/s)
  Call Extruder(999.07533)
  MoveL 3275 to (522.31, 444.19, 56) mm, rotated rx 180 ry 0 rz 160 deg; joints [-0.833, 72.835, -13.353, -158.026, 61.337, 169.046]
  Call Extruder(1006.07214)
  MoveL 3276 to (520.26, 443.42, 56) mm, rotated rx -180 ry 0 rz 160 deg; joints [-0.931, 72.505, -12.624, -158.216, 61.689, 169.268]
  Set speed (17.6 mm/s)
  Call Extruder(1013.22479)
  MoveL 3277 to (518.14, 442.7, 56) mm, rotated rx -180 ry 0 rz 160 deg; joints [-1.022, 72.168, -11.877, -158.4, 62.053, 169.488]
  Set speed (17.6 mm/s)
  Call Extruder(1020.06874)
  MoveL 3278 to (516.09, 442.09, 56) mm, rotated rx -180 ry 0 rz 160 deg; joints [-1.102, 71.847, -11.161, -158.564, 62.405, 169.693]
  Set speed (17.6 mm/s)
  Call Extruder(1027.96969)
  MoveL 3279 to (513.7, 441.48, 56) mm, rotated rx 180 ry 0 rz 160 deg; joints [-1.184, 71.477, -10.335, -158.741, 62.816, 169.921]
  Call Extruder(1034.32513)
  MoveL 3280 to (511.76, 441.06, 56) mm, rotated rx -180 ry 0 rz 160 deg; joints [-1.24, 71.18, -9.671, -158.871, 63.148, 170.099]
  Set speed (17.6 mm/s)
  Call Extruder(1041.32792)
  MoveL 3281 to (509.61, 440.67, 56) mm, rotated rx -180 ry 0 rz 160 deg; joints [-1.295, 70.855, -8.941, -159.005, 63.517, 170.289]
  Set speed (17.6 mm/s)
  Call Extruder(1048.47944)
  MoveL 3282 to (507.39, 440.36, 56) mm, rotated rx -180 ry 0 rz 160 deg; joints [-1.341, 70.526, -8.198, -159.128, 63.896, 170.476]
  Set speed (17.6 mm/s)
  Call Extruder(1055.70688)
  MoveL 3283 to (505.15, 440.12, 56) mm, rotated rx -180 ry 0 rz 160 deg; joints [-1.377, 70.195, -7.45, -159.24, 64.28, 170.658]
  Set speed (17.6 mm/s)
  Call Extruder(1062.72145)
  MoveL 3284 to (502.96, 439.97, 56) mm, rotated rx 180 ry 0 rz 160 deg; joints [-1.403, 69.877, -6.728, -159.336, 64.654, 170.829]
  Call Extruder(1069.86364)
  MoveL 3285 to (500.73, 439.9, 56) mm, rotated rx 180 ry 0 rz 160 deg; joints [-1.418, 69.557, -5.998, -159.421, 65.035, 170.995]
  Set speed (17.6 mm/s)
  Call Extruder(1076.83912)
  MoveL 3286 to (498.55, 439.92, 56) mm, rotated rx -180 ry 0 rz 160 deg; joints [-1.423, 69.248, -5.291, -159.491, 65.407, 171.151]
  Call Extruder(1084.02562)
  MoveL 3287 to (496.31, 440.01, 56) mm, rotated rx 180 ry 0 rz 160 deg; joints [-1.418, 68.933, -4.569, -159.55, 65.789, 171.306]
  Set speed (17.6 mm/s)
  Call Extruder(1090.96433)
  MoveL 3288 to (494.14, 440.19, 56) mm, rotated rx 180 ry 0 rz 160 deg; joints [-1.403, 68.634, -3.878, -159.594, 66.158, 171.448]
  Set speed (17.6 mm/s)
  Call Extruder(1098.54235)
  MoveL 3289 to (491.79, 440.46, 56) mm, rotated rx 180 ry 0 rz 160 deg; joints [-1.375, 68.312, -3.134, -159.628, 66.558, 171.597]
  Set speed (17.6 mm/s)
  Call Extruder(1105.29006)
  MoveL 3290 to (489.71, 440.78, 56) mm, rotated rx 180 ry 0 rz 160 deg; joints [-1.339, 68.03, -2.479, -159.645, 66.913, 171.723]
  Call Extruder(1112.20866)
  MoveL 3291 to (487.59, 441.19, 56) mm, rotated rx -180 ry 0 rz 160 deg; joints [-1.291, 67.746, -1.817, -159.65, 67.274, 171.846]
  Set speed (17.6 mm/s)
  Call Extruder(1119.28251)
  MoveL 3292 to (485.43, 441.69, 56) mm, rotated rx 180 ry 0 rz 160 deg; joints [-1.233, 67.461, -1.15, -159.642, 67.641, 171.965]
  Call Extruder(1126.52561)
  MoveL 3293 to (483.25, 442.28, 56) mm, rotated rx -180 ry 0 rz 160 deg; joints [-1.161, 67.175, -0.478, -159.62, 68.013, 172.081]
  Set speed (17.6 mm/s)
  Call Extruder(1133.57297)
  MoveL 3294 to (481.15, 442.93, 56) mm, rotated rx 180 ry 0 rz 160 deg; joints [-1.08, 66.903, 0.164, -159.585, 68.37, 172.188]
  Call Extruder(1140.69966)
  MoveL 3295 to (479.04, 443.67, 56) mm, rotated rx -180 ry 0 rz 160 deg; joints [-0.986, 66.634, 0.8, -159.536, 68.727, 172.29]
  Set speed (17.6 mm/s)
  Call Extruder(1147.65858)
  MoveL 3296 to (477.02, 444.46, 56) mm, rotated rx 180 ry 0 rz 160 deg; joints [-0.884, 66.378, 1.409, -159.475, 69.071, 172.383]
  Call Extruder(1154.78004)
  MoveL 3297 to (474.98, 445.35, 56) mm, rotated rx -180 ry 0 rz 160 deg; joints [-0.768, 66.123, 2.018, -159.4, 69.418, 172.472]
  Set speed (17.6 mm/s)
  Call Extruder(1161.00138)
  MoveL 3298 to (473.23, 446.18, 56) mm, rotated rx -180 ry 0 rz 160 deg; joints [-0.659, 65.905, 2.539, -159.324, 69.716, 172.546]
  Set speed (17.6 mm/s)
  Call Extruder(1168.89953)
  MoveL 3299 to (471.05, 447.33, 56) mm, rotated rx 180 ry 0 rz 160 deg; joints [-0.506, 65.638, 3.182, -159.211, 70.087, 172.632]
  Set speed (17.6 mm/s)
  Call Extruder(1176.03748)
  MoveL 3300 to (469.11, 448.44, 56) mm, rotated rx 180 ry 0 rz 160 deg; joints [-0.356, 65.404, 3.747, -159.095, 70.416, 172.704]
  Set speed (17.6 mm/s)
  Call Extruder(1183.21267)
  MoveL 3301 to (467.21, 449.63, 56) mm, rotated rx 180 ry 0 rz 160 deg; joints [-0.195, 65.176, 4.299, -158.966, 70.739, 172.771]
  Set speed (17.6 mm/s)
  Call Extruder(1190.78714)
  MoveL 3302 to (465.25, 450.96, 56) mm, rotated rx 180 ry 0 rz 160 deg; joints [-0.012, 64.945, 4.862, -158.816, 71.072, 172.835]
  Set speed (17.6 mm/s)
  Call Extruder(1197.04558)
  MoveL 3303 to (463.68, 452.11, 56) mm, rotated rx 180 ry 0 rz 160 deg; joints [0.148, 64.761, 5.312, -158.681, 71.339, 172.882]
  Set speed (17.6 mm/s)
  Call Extruder(1204.34815)
  MoveL 3304 to (461.89, 453.52, 56) mm, rotated rx -180 ry 0 rz 160 deg; joints [0.346, 64.554, 5.82, -158.511, 71.643, 172.932]
  Set speed (17.6 mm/s)
  Call Extruder(1211.55307)
  MoveL 3305 to (460.18, 454.98, 56) mm, rotated rx 180 ry 0 rz 160 deg; joints [0.551, 64.358, 6.301, -158.331, 71.935, 172.976]
  Set speed (17.6 mm/s)
  Call Extruder(1218.63143)
  MoveL 3306 to (458.55, 456.48, 56) mm, rotated rx 180 ry 0 rz 160 deg; joints [0.764, 64.175, 6.755, -158.141, 72.211, 173.013]
  Set speed (17.6 mm/s)
  Call Extruder(1225.56938)
  MoveL 3307 to (457.01, 458, 56) mm, rotated rx -180 ry 0 rz 160 deg; joints [0.981, 64.003, 7.181, -157.945, 72.473, 173.044]
  Set speed (17.6 mm/s)
  Call Extruder(1232.79742)
  MoveL 3308 to (455.46, 459.65, 56) mm, rotated rx 180 ry 0 rz 160 deg; joints [1.218, 63.833, 7.604, -157.729, 72.736, 173.07]
  Set speed (17.6 mm/s)
  Call Extruder(1239.88285)
  MoveL 3309 to (454, 461.31, 56) mm, rotated rx -180 ry 0 rz 160 deg; joints [1.459, 63.675, 7.997, -157.506, 72.983, 173.09]
  Set speed (17.6 mm/s)
  Call Extruder(1246.81848)
  MoveL 3310 to (452.64, 463, 56) mm, rotated rx 180 ry 0 rz 160 deg; joints [1.703, 63.529, 8.362, -157.278, 73.214, 173.104]
  Set speed (17.6 mm/s)
  Call Extruder(1254.04746)
  MoveL 3311 to (451.28, 464.8, 56) mm, rotated rx -180 ry 0 rz 160 deg; joints [1.967, 63.387, 8.72, -157.03, 73.444, 173.113]
  Set speed (17.6 mm/s)
  Call Extruder(1261.12658)
  MoveL 3312 to (450.02, 466.62, 56) mm, rotated rx 180 ry 0 rz 160 deg; joints [2.234, 63.256, 9.048, -156.777, 73.658, 173.116]
  Set speed (17.6 mm/s)
  Call Extruder(1268.06297)
  MoveL 3313 to (448.85, 468.44, 56) mm, rotated rx -180 ry 0 rz 160 deg; joints [2.503, 63.138, 9.347, -156.52, 73.857, 173.113]
  Set speed (17.6 mm/s)
  Call Extruder(1275.28258)
  MoveL 3314 to (447.7, 470.39, 56) mm, rotated rx -180 ry 0 rz 160 deg; joints [2.79, 63.024, 9.636, -156.243, 74.051, 173.104]
  Set speed (17.6 mm/s)
  Call Extruder(1282.32547)
  MoveL 3315 to (446.65, 472.32, 56) mm, rotated rx -180 ry 0 rz 160 deg; joints [3.076, 62.922, 9.895, -155.966, 74.229, 173.089]
  Set speed (17.6 mm/s)
  Call Extruder(1289.41145)
  MoveL 3316 to (445.67, 474.3, 56) mm, rotated rx 180 ry 0 rz 160 deg; joints [3.371, 62.829, 10.131, -155.678, 74.395, 173.068]
  Set speed (17.6 mm/s)
  Call Extruder(1297.25766)
  MoveL 3317 to (444.66, 476.54, 56) mm, rotated rx 180 ry 0 rz 160 deg; joints [3.703, 62.737, 10.364, -155.352, 74.564, 173.037]
  Set speed (17.6 mm/s)
  Call Extruder(1303.63583)
  MoveL 3318 to (443.92, 478.38, 56) mm, rotated rx 180 ry 0 rz 160 deg; joints [3.978, 62.671, 10.532, -155.081, 74.69, 173.007]
  Set speed (17.6 mm/s)
  Call Extruder(1310.70619)
  MoveL 3319 to (443.16, 480.46, 56) mm, rotated rx 180 ry 0 rz 160 deg; joints [4.287, 62.608, 10.695, -154.775, 74.818, 172.967]
  Set speed (17.6 mm/s)
  Call Extruder(1317.78489)
  MoveL 3320 to (442.48, 482.57, 56) mm, rotated rx 180 ry 0 rz 160 deg; joints [4.6, 62.554, 10.834, -154.462, 74.933, 172.92]
  Set speed (17.6 mm/s)
  Call Extruder(1324.86671)
  MoveL 3321 to (441.88, 484.69, 56) mm, rotated rx 180 ry 0 rz 160 deg; joints [4.917, 62.509, 10.949, -154.145, 75.035, 172.867]
  Set speed (17.6 mm/s)
  Call Extruder(1331.94242)
  MoveL 3322 to (441.35, 486.84, 56) mm, rotated rx 180 ry 0 rz 160 deg; joints [5.236, 62.474, 11.037, -153.823, 75.124, 172.807]
  Set speed (17.6 mm/s)
  Call Extruder(1338.88118)
  MoveL 3323 to (440.92, 488.97, 56) mm, rotated rx -180 ry 0 rz 160 deg; joints [5.551, 62.45, 11.1, -153.505, 75.198, 172.742]
  Set speed (17.6 mm/s)
  Call Extruder(1346.11264)
  MoveL 3324 to (440.55, 491.19, 56) mm, rotated rx 180 ry 0 rz 160 deg; joints [5.881, 62.434, 11.141, -153.17, 75.262, 172.668]
  Set speed (17.6 mm/s)
  Call Extruder(1353.19822)
  MoveL 3325 to (440.26, 493.39, 56) mm, rotated rx -180 ry 0 rz 160 deg; joints [6.204, 62.429, 11.154, -152.839, 75.31, 172.587]
  Call Extruder(1360.27824)
  MoveL 3326 to (440.06, 495.59, 56) mm, rotated rx -180 ry 0 rz 160 deg; joints [6.527, 62.433, 11.143, -152.507, 75.346, 172.5]
  Set speed (17.6 mm/s)
  Call Extruder(1367.28463)
  MoveL 3327 to (439.94, 497.78, 56) mm, rotated rx -180 ry 0 rz 160 deg; joints [6.847, 62.447, 11.107, -152.177, 75.369, 172.407]
  Call Extruder(1374.44497)
  MoveL 3328 to (439.9, 500.01, 56) mm, rotated rx 180 ry 0 rz 160 deg; joints [7.172, 62.471, 11.045, -151.839, 75.378, 172.304]
  Set speed (17.6 mm/s)
  Call Extruder(1382.32415)
  MoveL 3329 to (439.95, 502.48, 56) mm, rotated rx -180 ry 0 rz 160 deg; joints [7.527, 62.51, 10.946, -151.468, 75.374, 172.183]
  Set speed (17.6 mm/s)
  Call Extruder(1390.08998)
  MoveL 3330 to (440.1, 504.9, 56) mm, rotated rx 180 ry 0 rz 160 deg; joints [7.874, 62.559, 10.819, -151.103, 75.353, 172.055]
  Set speed (17.6 mm/s)
  Call Extruder(1397.96651)
  MoveL 3331 to (440.35, 507.34, 56) mm, rotated rx -180 ry 0 rz 160 deg; joints [8.222, 62.621, 10.66, -150.735, 75.317, 171.916]
  Set speed (17.6 mm/s)
  Call Extruder(1405.83454)
  MoveL 3332 to (440.7, 509.78, 56) mm, rotated rx 180 ry 0 rz 160 deg; joints [8.565, 62.696, 10.471, -150.369, 75.265, 171.768]
  Set speed (17.6 mm/s)
  Call Extruder(1413.75943)
  MoveL 3333 to (441.15, 512.21, 56) mm, rotated rx -180 ry 0 rz 160 deg; joints [8.904, 62.782, 10.249, -150.004, 75.198, 171.61]
  Set speed (17.6 mm/s)
  Call Extruder(1417.69355)
  MoveL 3334 to (441.42, 513.41, 56) mm, rotated rx -180 ry 0 rz 160 deg; joints [9.069, 62.83, 10.127, -149.825, 75.157, 171.529]
  Set speed (17.6 mm/s)
  Call Extruder(1421.67738)
  MoveL 3335 to (441.7, 514.62, 56) mm, rotated rx -180 ry 0 rz 160 deg; joints [9.236, 62.881, 9.999, -149.644, 75.115, 171.444]
  Set speed (17.6 mm/s)
  Call Extruder(1429.37707)
  MoveL 3336 to (442.33, 516.94, 56) mm, rotated rx 180 ry 0 rz 160 deg; joints [9.552, 62.988, 9.727, -149.299, 75.02, 171.274]
  Set speed (17.6 mm/s)
  Call Extruder(1433.41205)
  MoveL 3337 to (442.71, 518.14, 56) mm, rotated rx 180 ry 0 rz 160 deg; joints [9.714, 63.049, 9.571, -149.12, 74.964, 171.182]
  Set speed (17.6 mm/s)
  Call Extruder(1437.40864)
  MoveL 3338 to (443.09, 519.33, 56) mm, rotated rx 180 ry 0 rz 160 deg; joints [9.872, 63.112, 9.413, -148.945, 74.906, 171.088]
  Set speed (17.6 mm/s)
  Call Extruder(1441.80714)
  MoveL 3339 to (443.55, 520.62, 56) mm, rotated rx -180 ry 0 rz 160 deg; joints [10.044, 63.185, 9.228, -148.753, 74.838, 170.983]
  Call Extruder(1445.23697)
  MoveL 3340 to (443.92, 521.62, 56) mm, rotated rx -180 ry 0 rz 160 deg; joints [10.176, 63.244, 9.08, -148.605, 74.782, 170.899]
  Set speed (17.6 mm/s)
  Call Extruder(1449.18479)
  MoveL 3341 to (444.38, 522.77, 56) mm, rotated rx 180 ry 0 rz 160 deg; joints [10.326, 63.315, 8.9, -148.437, 74.713, 170.8]
  Set speed (17.6 mm/s)
  Call Extruder(1453.07262)
  MoveL 3342 to (444.85, 523.89, 56) mm, rotated rx 180 ry 0 rz 160 deg; joints [10.471, 63.387, 8.719, -148.272, 74.643, 170.701]
  Set speed (17.6 mm/s)
  Call Extruder(1459.94055)
  MoveL 3343 to (445.74, 525.84, 56) mm, rotated rx 180 ry 0 rz 160 deg; joints [10.721, 63.522, 8.379, -147.987, 74.511, 170.521]
  Set speed (17.6 mm/s)
  Call Extruder(1464.83455)
  MoveL 3344 to (446.41, 527.21, 56) mm, rotated rx 180 ry 0 rz 160 deg; joints [10.895, 63.624, 8.125, -147.786, 74.41, 170.389]
  Set speed (17.6 mm/s)
  Call Extruder(1468.88609)
  MoveL 3345 to (446.99, 528.33, 56) mm, rotated rx 180 ry 0 rz 160 deg; joints [11.036, 63.711, 7.907, -147.622, 74.323, 170.278]
  Set speed (17.6 mm/s)
  Call Extruder(1472.81871)
  MoveL 3346 to (447.58, 529.41, 56) mm, rotated rx 180 ry 0 rz 160 deg; joints [11.17, 63.799, 7.688, -147.466, 74.235, 170.168]
  Call Extruder(1476.69401)
  MoveL 3347 to (448.18, 530.46, 56) mm, rotated rx 180 ry 0 rz 160 deg; joints [11.299, 63.888, 7.467, -147.313, 74.146, 170.058]
  Set speed (17.6 mm/s)
  Call Extruder(1480.61322)
  MoveL 3348 to (448.81, 531.51, 56) mm, rotated rx -180 ry 0 rz 160 deg; joints [11.427, 63.98, 7.237, -147.161, 74.053, 169.944]
  Set speed (17.6 mm/s)
  Call Extruder(1484.53546)
  MoveL 3349 to (449.47, 532.54, 56) mm, rotated rx 180 ry 0 rz 160 deg; joints [11.551, 64.076, 7, -147.011, 73.956, 169.829]
  Set speed (17.6 mm/s)
  Call Extruder(1488.43566)
  MoveL 3350 to (450.14, 533.56, 56) mm, rotated rx -180 ry 0 rz 160 deg; joints [11.673, 64.173, 6.758, -146.865, 73.857, 169.713]
  Set speed (17.6 mm/s)
  Call Extruder(1492.53278)
  MoveL 3351 to (450.86, 534.62, 56) mm, rotated rx -180 ry 0 rz 160 deg; joints [11.797, 64.279, 6.498, -146.713, 73.749, 169.589]
  Set speed (17.6 mm/s)
  Call Extruder(1496.35689)
  MoveL 3352 to (451.57, 535.58, 56) mm, rotated rx -180 ry 0 rz 160 deg; joints [11.91, 64.38, 6.248, -146.573, 73.646, 169.472]
  Set speed (17.6 mm/s)
  Call Extruder(1500.24847)
  MoveL 3353 to (452.29, 536.56, 56) mm, rotated rx -180 ry 0 rz 160 deg; joints [12.022, 64.485, 5.99, -146.434, 73.538, 169.351]
  Set speed (17.6 mm/s)
  Call Extruder(1504.28322)
  MoveL 3354 to (453.07, 537.55, 56) mm, rotated rx 180 ry 0 rz 160 deg; joints [12.134, 64.596, 5.716, -146.291, 73.424, 169.224]
  Call Extruder(1508.13248)
  MoveL 3355 to (453.83, 538.48, 56) mm, rotated rx -180 ry 0 rz 160 deg; joints [12.238, 64.705, 5.448, -146.158, 73.312, 169.102]
  Set speed (17.6 mm/s)
  Call Extruder(1512.11069)
  MoveL 3356 to (454.64, 539.43, 56) mm, rotated rx 180 ry 0 rz 160 deg; joints [12.343, 64.821, 5.166, -146.023, 73.193, 168.973]
  Set speed (17.6 mm/s)
  Call Extruder(1516.14085)
  MoveL 3357 to (455.47, 540.37, 56) mm, rotated rx 180 ry 0 rz 160 deg; joints [12.446, 64.94, 4.874, -145.889, 73.07, 168.842]
  Set speed (17.6 mm/s)
  Call Extruder(1520.00041)
  MoveL 3358 to (456.29, 541.25, 56) mm, rotated rx -180 ry 0 rz 160 deg; joints [12.54, 65.057, 4.59, -145.763, 72.95, 168.715]
  Set speed (17.6 mm/s)
  Call Extruder(1523.86177)
  MoveL 3359 to (457.13, 542.12, 56) mm, rotated rx -180 ry 0 rz 160 deg; joints [12.632, 65.176, 4.3, -145.639, 72.827, 168.587]
  Set speed (17.6 mm/s)
  Call Extruder(1527.81594)
  MoveL 3360 to (458, 543, 56) mm, rotated rx 180 ry 0 rz 160 deg; joints [12.723, 65.3, 3.998, -145.515, 72.699, 168.454]
  Set speed (17.6 mm/s)
  Call Extruder(1531.87366)
  MoveL 3361 to (458.92, 543.87, 56) mm, rotated rx -180 ry 0 rz 160 deg; joints [12.812, 65.43, 3.683, -145.39, 72.564, 168.317]
  Set speed (17.6 mm/s)
  Call Extruder(1535.75393)
  MoveL 3362 to (459.81, 544.69, 56) mm, rotated rx -180 ry 0 rz 160 deg; joints [12.894, 65.557, 3.377, -145.274, 72.433, 168.185]
  Set speed (17.6 mm/s)
  Call Extruder(1539.63013)
  MoveL 3363 to (460.72, 545.49, 56) mm, rotated rx -180 ry 0 rz 160 deg; joints [12.973, 65.686, 3.066, -145.16, 72.3, 168.051]
  Set speed (17.6 mm/s)
  Call Extruder(1543.55201)
  MoveL 3364 to (461.66, 546.28, 56) mm, rotated rx 180 ry 0 rz 160 deg; joints [13.049, 65.819, 2.747, -145.048, 72.163, 167.915]
  Call Extruder(1547.47285)
  MoveL 3365 to (462.61, 547.06, 56) mm, rotated rx -180 ry 0 rz 160 deg; joints [13.122, 65.954, 2.423, -144.938, 72.024, 167.778]
  Set speed (17.6 mm/s)
  Call Extruder(1551.49559)
  MoveL 3366 to (463.6, 547.83, 56) mm, rotated rx -180 ry 0 rz 160 deg; joints [13.192, 66.094, 2.086, -144.828, 71.878, 167.637]
  Set speed (17.6 mm/s)
  Call Extruder(1555.36925)
  MoveL 3367 to (464.57, 548.55, 56) mm, rotated rx 180 ry 0 rz 160 deg; joints [13.258, 66.232, 1.757, -144.725, 71.736, 167.5]
  Call Extruder(1559.33543)
  MoveL 3368 to (465.58, 549.27, 56) mm, rotated rx -180 ry 0 rz 160 deg; joints [13.321, 66.375, 1.416, -144.622, 71.588, 167.359]
  Set speed (17.6 mm/s)
  Call Extruder(1563.29773)
  MoveL 3369 to (466.6, 549.97, 56) mm, rotated rx -180 ry 0 rz 160 deg; joints [13.38, 66.52, 1.071, -144.522, 71.438, 167.217]
  Set speed (17.6 mm/s)
  Call Extruder(1567.21475)
  MoveL 3370 to (467.63, 550.64, 56) mm, rotated rx -180 ry 0 rz 160 deg; joints [13.436, 66.665, 0.726, -144.426, 71.288, 167.077]
  Set speed (17.6 mm/s)
  Call Extruder(1570.44196)
  MoveL 3371 to (468.48, 551.18, 56) mm, rotated rx -180 ry 0 rz 160 deg; joints [13.479, 66.787, 0.438, -144.349, 71.162, 166.96]
  Call Extruder(0.00000)
  Set speed (17.6 mm/s)
  Call Extruder(4.04830)
  MoveL 3372 to (469.56, 551.83, 56) mm, rotated rx -180 ry 0 rz 160 deg; joints [13.53, 66.941, 0.074, -144.254, 71.003, 166.813]
  Set speed (17.6 mm/s)
  Call Extruder(8.55195)
  MoveL 3373 to (470.78, 552.53, 56) mm, rotated rx -180 ry 0 rz 160 deg; joints [13.582, 67.114, -0.336, -144.153, 70.824, 166.65]
  Set speed (17.6 mm/s)
  Call Extruder(13.62488)
  MoveL 3374 to (472.18, 553.28, 56) mm, rotated rx -180 ry 0 rz 160 deg; joints [13.635, 67.313, -0.803, -144.043, 70.618, 166.465]
  Set speed (17.6 mm/s)
  Call Extruder(16.38174)
  MoveL 3375 to (472.94, 553.67, 56) mm, rotated rx 180 ry 0 rz 160 deg; joints [13.662, 67.422, -1.059, -143.985, 70.506, 166.364]
  Call Extruder(20.35440)
  MoveL 3376 to (474.06, 554.22, 56) mm, rotated rx -180 ry 0 rz 160 deg; joints [13.697, 67.581, -1.431, -143.904, 70.341, 166.219]
  Set speed (17.6 mm/s)
  Call Extruder(25.29476)
  MoveL 3377 to (475.46, 554.87, 56) mm, rotated rx -180 ry 0 rz 160 deg; joints [13.736, 67.781, -1.899, -143.807, 70.135, 166.037]
  Set speed (17.6 mm/s)
  Call Extruder(32.14947)
  MoveL 3378 to (477.42, 555.71, 56) mm, rotated rx 180 ry 0 rz 160 deg; joints [13.781, 68.062, -2.555, -143.68, 69.844, 165.785]
  Set speed (17.6 mm/s)
  Call Extruder(36.17617)
  MoveL 3379 to (478.6, 556.16, 56) mm, rotated rx 180 ry 0 rz 160 deg; joints [13.802, 68.23, -2.945, -143.609, 69.67, 165.638]
  Set speed (17.6 mm/s)
  Call Extruder(40.21620)
  MoveL 3380 to (479.78, 556.6, 56) mm, rotated rx -180 ry 0 rz 160 deg; joints [13.822, 68.4, -3.339, -143.54, 69.495, 165.489]
  Call Extruder(44.08218)
  MoveL 3381 to (480.92, 556.99, 56) mm, rotated rx 180 ry 0 rz 160 deg; joints [13.835, 68.564, -3.719, -143.478, 69.325, 165.347]
  Set speed (17.6 mm/s)
  Call Extruder(48.09152)
  MoveL 3382 to (482.11, 557.38, 56) mm, rotated rx -180 ry 0 rz 160 deg; joints [13.847, 68.736, -4.115, -143.415, 69.147, 165.199]
  Set speed (17.6 mm/s)
  Call Extruder(55.95660)
  MoveL 3383 to (484.47, 558.06, 56) mm, rotated rx -180 ry 0 rz 160 deg; joints [13.86, 69.077, -4.9, -143.3, 68.795, 164.911]
  Set speed (17.6 mm/s)
  Call Extruder(59.79459)
  MoveL 3384 to (485.63, 558.35, 56) mm, rotated rx -180 ry 0 rz 160 deg; joints [13.861, 69.245, -5.286, -143.248, 68.62, 164.771]
  Set speed (17.6 mm/s)
  Call Extruder(63.65458)
  MoveL 3385 to (486.8, 558.64, 56) mm, rotated rx 180 ry 0 rz 160 deg; joints [13.86, 69.416, -5.675, -143.198, 68.444, 164.63]
  Set speed (17.6 mm/s)
  Call Extruder(71.68423)
  MoveL 3386 to (489.26, 559.14, 56) mm, rotated rx -180 ry 0 rz 160 deg; joints [13.847, 69.774, -6.493, -143.101, 68.073, 164.338]
  Set speed (17.6 mm/s)
  Call Extruder(79.51788)
  MoveL 3387 to (491.67, 559.53, 56) mm, rotated rx 180 ry 0 rz 160 deg; joints [13.821, 70.128, -7.298, -143.017, 67.706, 164.056]
  Call Extruder(87.31778)
  MoveL 3388 to (494.09, 559.81, 56) mm, rotated rx 180 ry 0 rz 160 deg; joints [13.784, 70.484, -8.104, -142.944, 67.336, 163.778]
  Set speed (17.6 mm/s)
  Call Extruder(95.11340)
  MoveL 3389 to (496.52, 560, 56) mm, rotated rx 180 ry 0 rz 160 deg; joints [13.734, 70.843, -8.914, -142.881, 66.963, 163.503]
  Call Extruder(103.14389)
  MoveL 3390 to (499.03, 560.1, 56) mm, rotated rx -180 ry 0 rz 160 deg; joints [13.672, 71.216, -9.752, -142.826, 66.574, 163.223]
  Set speed (10.0 mm/s)
  MoveL 3391 to (499.03, 560.1, 60) mm, rotated rx -180 ry 0 rz 160 deg; joints [13.672, 70.53, -9.328, -142.757, 66.365, 163.05]
  Set speed (120.0 mm/s)
  MoveL 3392 to (499.01, 560.9, 60) mm, rotated rx 180 ry 0 rz 160 deg; joints [13.77, 70.557, -9.389, -142.646, 66.367, 162.987]
  Set speed (17.7 mm/s)
  Call Extruder(111.16027)
  MoveL 3393 to (496.51, 560.81, 60) mm, rotated rx 180 ry 0 rz 160 deg; joints [13.833, 70.183, -8.553, -142.701, 66.753, 163.266]
  Set speed (17.7 mm/s)
  Call Extruder(119.15182)
  MoveL 3394 to (494.01, 560.62, 60) mm, rotated rx -180 ry 0 rz 160 deg; joints [13.884, 69.813, -7.723, -142.767, 67.133, 163.547]
  Set speed (17.7 mm/s)
  Call Extruder(127.04156)
  MoveL 3395 to (491.56, 560.32, 60) mm, rotated rx 180 ry 0 rz 160 deg; joints [13.922, 69.451, -6.909, -142.841, 67.504, 163.828]
  Set speed (17.7 mm/s)
  Call Extruder(134.91434)
  MoveL 3396 to (489.13, 559.93, 60) mm, rotated rx 180 ry 0 rz 160 deg; joints [13.948, 69.094, -6.101, -142.925, 67.871, 164.112]
  Call Extruder(143.07304)
  MoveL 3397 to (486.63, 559.42, 60) mm, rotated rx 180 ry 0 rz 160 deg; joints [13.963, 68.728, -5.271, -143.023, 68.245, 164.408]
  Set speed (17.6 mm/s)
  Call Extruder(146.99918)
  MoveL 3398 to (485.43, 559.14, 60) mm, rotated rx 180 ry 0 rz 160 deg; joints [13.964, 68.554, -4.874, -143.075, 68.423, 164.551]
  Set speed (17.6 mm/s)
  Call Extruder(150.81418)
  MoveL 3399 to (484.28, 558.85, 60) mm, rotated rx 180 ry 0 rz 160 deg; joints [13.963, 68.386, -4.491, -143.126, 68.595, 164.69]
  Call Extruder(154.92140)
  MoveL 3400 to (483.04, 558.5, 60) mm, rotated rx 180 ry 0 rz 160 deg; joints [13.958, 68.206, -4.081, -143.186, 68.778, 164.841]
  Set speed (17.6 mm/s)
  Call Extruder(158.85012)
  MoveL 3401 to (481.87, 558.15, 60) mm, rotated rx -180 ry 0 rz 160 deg; joints [13.951, 68.036, -3.69, -143.244, 68.953, 164.985]
  Set speed (17.6 mm/s)
  Call Extruder(167.04979)
  MoveL 3402 to (479.44, 557.33, 60) mm, rotated rx -180 ry 0 rz 160 deg; joints [13.925, 67.684, -2.883, -143.375, 69.312, 165.286]
  Set speed (17.6 mm/s)
  Call Extruder(174.70417)
  MoveL 3403 to (477.2, 556.48, 60) mm, rotated rx -180 ry 0 rz 160 deg; joints [13.887, 67.361, -2.139, -143.508, 69.64, 165.567]
  Set speed (17.6 mm/s)
  Call Extruder(178.86993)
  MoveL 3404 to (476, 555.98, 60) mm, rotated rx -180 ry 0 rz 160 deg; joints [13.86, 67.188, -1.739, -143.585, 69.816, 165.721]
  Call Extruder(182.64118)
  MoveL 3405 to (474.92, 555.5, 60) mm, rotated rx -180 ry 0 rz 160 deg; joints [13.834, 67.033, -1.38, -143.657, 69.975, 165.859]
  Set speed (17.7 mm/s)
  Call Extruder(186.85594)
  MoveL 3406 to (473.72, 554.95, 60) mm, rotated rx 180 ry 0 rz 160 deg; joints [13.801, 66.862, -0.981, -143.739, 70.15, 166.014]
  Set speed (17.7 mm/s)
  Call Extruder(190.79866)
  MoveL 3407 to (472.61, 554.41, 60) mm, rotated rx 180 ry 0 rz 160 deg; joints [13.766, 66.703, -0.611, -143.82, 70.311, 166.158]
  Set speed (17.6 mm/s)
  Call Extruder(194.70590)
  MoveL 3408 to (471.53, 553.85, 60) mm, rotated rx 180 ry 0 rz 160 deg; joints [13.729, 66.547, -0.249, -143.903, 70.47, 166.301]
  Call Extruder(198.67956)
  MoveL 3409 to (470.44, 553.26, 60) mm, rotated rx 180 ry 0 rz 160 deg; joints [13.687, 66.391, 0.117, -143.989, 70.629, 166.446]
  Set speed (17.7 mm/s)
  Call Extruder(202.62893)
  MoveL 3410 to (469.36, 552.64, 60) mm, rotated rx -180 ry 0 rz 160 deg; joints [13.641, 66.238, 0.476, -144.079, 70.785, 166.59]
  Call Extruder(206.75063)
  MoveL 3411 to (468.25, 551.98, 60) mm, rotated rx 180 ry 0 rz 160 deg; joints [13.591, 66.08, 0.848, -144.174, 70.946, 166.739]
  Set speed (17.7 mm/s)
  Call Extruder(210.63738)
  MoveL 3412 to (467.22, 551.34, 60) mm, rotated rx -180 ry 0 rz 160 deg; joints [13.539, 65.932, 1.194, -144.267, 71.096, 166.879]
  Set speed (17.7 mm/s)
  Call Extruder(214.62750)
  MoveL 3413 to (466.18, 550.66, 60) mm, rotated rx -180 ry 0 rz 160 deg; joints [13.483, 65.783, 1.546, -144.365, 71.248, 167.023]
  Call Extruder(218.59116)
  MoveL 3414 to (465.15, 549.96, 60) mm, rotated rx -180 ry 0 rz 160 deg; joints [13.424, 65.637, 1.891, -144.465, 71.397, 167.165]
  Set speed (17.7 mm/s)
  Call Extruder(222.58425)
  MoveL 3415 to (464.13, 549.23, 60) mm, rotated rx 180 ry 0 rz 160 deg; joints [13.361, 65.492, 2.235, -144.569, 71.544, 167.307]
  Set speed (17.7 mm/s)
  Call Extruder(226.73722)
  MoveL 3416 to (463.09, 548.46, 60) mm, rotated rx 180 ry 0 rz 160 deg; joints [13.291, 65.343, 2.588, -144.68, 71.696, 167.454]
  Set speed (17.7 mm/s)
  Call Extruder(230.50837)
  MoveL 3417 to (462.16, 547.73, 60) mm, rotated rx 180 ry 0 rz 160 deg; joints [13.225, 65.21, 2.903, -144.783, 71.831, 167.587]
  Call Extruder(234.55731)
  MoveL 3418 to (461.18, 546.93, 60) mm, rotated rx -180 ry 0 rz 160 deg; joints [13.15, 65.07, 3.238, -144.897, 71.973, 167.728]
  Call Extruder(238.51060)
  MoveL 3419 to (460.23, 546.14, 60) mm, rotated rx -180 ry 0 rz 160 deg; joints [13.073, 64.935, 3.56, -145.01, 72.11, 167.865]
  Set speed (17.7 mm/s)
  Call Extruder(242.46468)
  MoveL 3420 to (459.3, 545.32, 60) mm, rotated rx -180 ry 0 rz 160 deg; joints [12.993, 64.803, 3.877, -145.126, 72.245, 168.002]
  Call Extruder(246.47401)
